Yaskawa INFORM job: DEMO_ROOF_UPPER_0625_3PAINT_42.JBI

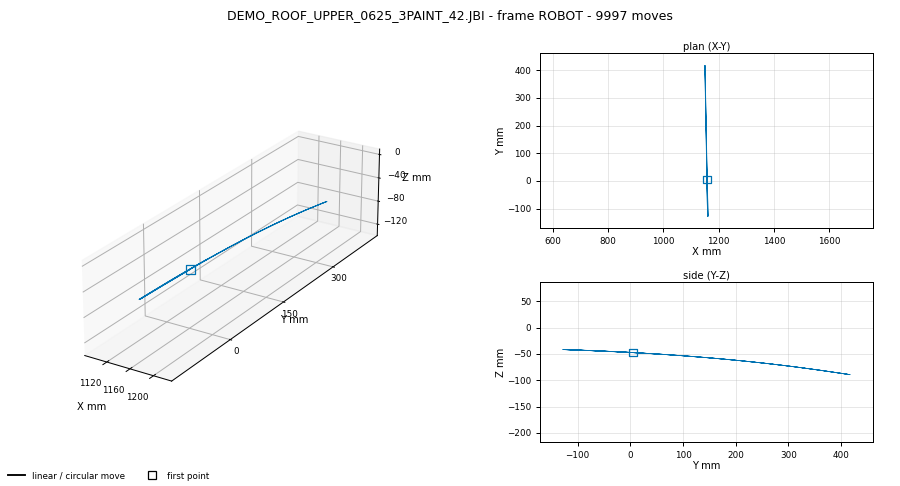
[picture p0: tool path of DEMO_ROOF_UPPER_0625_3PAINT_42.JBI in frame ROBOT, 9997 of 9997 moves have a stored position in this frame; points joined in program order, loops and branches not executed]
/JOB
//NAME DEMO_ROOF_UPPER_0625_3PAINT42
//POS
///NPOS 9997,0,0,0,0,0
///TOOL 0
///USER 0
///POSTYPE ROBOT
///RECTAN
///RCONF 1,0,0,0,0,0,0,0,0,0,0,0,0,0,0,0,0,0,0,0,0,0,0,0
C00000=1159.229,5.390,-47.328,179.872,6.067,149.128
C00001=1159.234,5.140,-47.313,179.870,6.066,149.128
C00002=1159.239,4.891,-47.300,179.867,6.066,149.129
C00003=1159.244,4.641,-47.286,179.865,6.065,149.129
C00004=1159.249,4.391,-47.273,179.863,6.064,149.130
C00005=1159.255,4.142,-47.259,179.860,6.063,149.131
C00006=1159.259,3.892,-47.246,179.858,6.063,149.131
C00007=1159.265,3.643,-47.232,179.855,6.061,149.132
C00008=1159.270,3.393,-47.218,179.852,6.061,149.132
C00009=1159.275,3.144,-47.205,179.850,6.060,149.133
C00010=1159.280,2.894,-47.192,179.848,6.060,149.134
C00011=1159.285,2.645,-47.178,179.845,6.059,149.134
C00012=1159.290,2.395,-47.165,179.843,6.058,149.135
C00013=1159.295,2.125,-47.150,179.840,6.058,149.135
C00014=1159.301,1.856,-47.135,179.837,6.057,149.136
C00015=1159.306,1.587,-47.121,179.835,6.056,149.137
C00016=1159.312,1.317,-47.106,179.832,6.055,149.137
C00017=1159.318,1.068,-47.093,179.829,6.055,149.138
C00018=1159.322,0.818,-47.080,179.827,6.054,149.138
C00019=1159.328,0.569,-47.066,179.824,6.053,149.139
C00020=1159.332,0.319,-47.053,179.822,6.052,149.140
C00021=1159.338,0.070,-47.039,179.819,6.052,149.140
C00022=1159.342,-0.180,-47.026,179.817,6.051,149.141
C00023=1159.348,-0.429,-47.013,179.814,6.050,149.141
C00024=1159.353,-0.680,-46.999,179.812,6.050,149.142
C00025=1159.358,-0.929,-46.986,179.809,6.049,149.143
C00026=1159.363,-1.179,-46.972,179.807,6.048,149.143
C00027=1159.368,-1.428,-46.960,179.805,6.048,149.144
C00028=1159.374,-1.678,-46.946,179.802,6.047,149.144
C00029=1159.379,-1.927,-46.933,179.799,6.046,149.145
C00030=1159.384,-2.177,-46.919,179.797,6.045,149.146
C00031=1159.389,-2.427,-46.906,179.794,6.044,149.146
C00032=1159.394,-2.676,-46.893,179.792,6.044,149.147
C00033=1159.399,-2.926,-46.880,179.790,6.043,149.147
C00034=1159.405,-3.175,-46.866,179.787,6.043,149.148
C00035=1159.410,-3.425,-46.854,179.785,6.042,149.148
C00036=1159.414,-3.674,-46.840,179.782,6.042,149.149
C00037=1159.420,-3.924,-46.827,179.780,6.041,149.150
C00038=1159.425,-4.174,-46.814,179.777,6.040,149.150
C00039=1159.430,-4.423,-46.801,179.775,6.039,149.151
C00040=1159.435,-4.673,-46.787,179.772,6.039,149.151
C00041=1159.441,-4.922,-46.774,179.770,6.039,149.152
C00042=1159.446,-5.172,-46.761,179.767,6.037,149.153
C00043=1159.450,-5.422,-46.748,179.764,6.036,149.153
C00044=1159.456,-5.671,-46.735,179.762,6.036,149.154
C00045=1159.460,-5.921,-46.721,179.759,6.035,149.154
C00046=1159.466,-6.170,-46.708,179.757,6.034,149.155
C00047=1159.471,-6.420,-46.696,179.755,6.034,149.156
C00048=1159.476,-6.670,-46.683,179.752,6.033,149.156
C00049=1159.482,-6.919,-46.669,179.750,6.033,149.157
C00050=1159.487,-7.169,-46.657,179.748,6.032,149.157
C00051=1159.492,-7.419,-46.643,179.745,6.031,149.158
C00052=1159.497,-7.668,-46.630,179.743,6.031,149.158
C00053=1159.502,-7.917,-46.617,179.740,6.030,149.159
C00054=1159.507,-8.167,-46.604,179.738,6.030,149.160
C00055=1159.512,-8.417,-46.591,179.735,6.029,149.160
C00056=1159.517,-8.667,-46.578,179.733,6.028,149.161
C00057=1159.523,-8.916,-46.565,179.731,6.028,149.161
C00058=1159.528,-9.166,-46.552,179.728,6.027,149.162
C00059=1159.532,-9.416,-46.540,179.726,6.026,149.162
C00060=1159.538,-9.665,-46.526,179.722,6.025,149.163
C00061=1159.543,-9.915,-46.514,179.720,6.024,149.164
C00062=1159.548,-10.165,-46.501,179.718,6.024,149.164
C00063=1159.554,-10.414,-46.488,179.715,6.023,149.165
C00064=1159.559,-10.664,-46.475,179.713,6.023,149.165
C00065=1159.564,-10.913,-46.462,179.711,6.022,149.166
C00066=1159.569,-11.163,-46.449,179.708,6.021,149.167
C00067=1159.574,-11.413,-46.436,179.705,6.021,149.167
C00068=1159.579,-11.662,-46.424,179.703,6.020,149.168
C00069=1159.584,-11.912,-46.411,179.700,6.020,149.168
C00070=1159.589,-12.161,-46.398,179.698,6.019,149.169
C00071=1159.595,-12.411,-46.385,179.696,6.018,149.170
C00072=1159.600,-12.661,-46.372,179.693,6.018,149.170
C00073=1159.605,-12.910,-46.359,179.691,6.017,149.171
C00074=1159.610,-13.159,-46.347,179.689,6.016,149.171
C00075=1159.616,-13.409,-46.333,179.686,6.016,149.172
C00076=1159.620,-13.659,-46.320,179.684,6.015,149.172
C00077=1159.625,-13.908,-46.308,179.681,6.015,149.173
C00078=1159.630,-14.158,-46.295,179.679,6.014,149.174
C00079=1159.636,-14.407,-46.283,179.676,6.013,149.174
C00080=1159.641,-14.657,-46.269,179.674,6.013,149.175
C00081=1159.646,-14.907,-46.257,179.671,6.012,149.175
C00082=1159.651,-15.157,-46.245,179.669,6.012,149.176
C00083=1159.656,-15.406,-46.232,179.667,6.011,149.177
C00084=1159.661,-15.656,-46.219,179.664,6.010,149.177
C00085=1159.667,-15.906,-46.206,179.662,6.010,149.178
C00086=1159.672,-16.155,-46.193,179.659,6.009,149.178
C00087=1159.677,-16.404,-46.181,179.657,6.008,149.179
C00088=1159.683,-16.654,-46.169,179.654,6.008,149.180
C00089=1159.687,-16.904,-46.156,179.652,6.007,149.180
C00090=1159.692,-17.154,-46.143,179.649,6.007,149.181
C00091=1159.697,-17.403,-46.131,179.647,6.006,149.181
C00092=1159.703,-17.652,-46.117,179.645,6.006,149.182
C00093=1159.708,-17.903,-46.105,179.642,6.005,149.183
C00094=1159.713,-18.152,-46.093,179.640,6.004,149.183
C00095=1159.718,-18.402,-46.080,179.637,6.004,149.184
C00096=1159.723,-18.651,-46.067,179.635,6.003,149.184
C00097=1159.728,-18.900,-46.055,179.632,6.003,149.185
C00098=1159.734,-19.150,-46.043,179.630,6.002,149.185
C00099=1159.738,-19.400,-46.030,179.627,6.001,149.186
C00100=1159.744,-19.650,-46.017,179.625,6.001,149.187
C00101=1159.750,-19.900,-46.005,179.623,6.000,149.187
C00102=1159.755,-20.149,-45.992,179.620,5.999,149.188
C00103=1159.760,-20.399,-45.980,179.618,5.999,149.188
C00104=1159.765,-20.648,-45.967,179.616,5.998,149.189
C00105=1159.770,-20.899,-45.955,179.613,5.998,149.190
C00106=1159.775,-21.148,-45.942,179.611,5.997,149.190
C00107=1159.780,-21.397,-45.930,179.608,5.996,149.191
C00108=1159.786,-21.647,-45.918,179.605,5.996,149.191
C00109=1159.791,-21.896,-45.905,179.603,5.995,149.192
C00110=1159.796,-22.146,-45.893,179.601,5.995,149.193
C00111=1159.801,-22.396,-45.881,179.598,5.994,149.193
C00112=1159.806,-22.645,-45.868,179.596,5.993,149.194
C00113=1159.811,-22.896,-45.856,179.594,5.993,149.194
C00114=1159.816,-23.145,-45.843,179.591,5.992,149.195
C00115=1159.821,-23.394,-45.831,179.589,5.991,149.195
C00116=1159.827,-23.644,-45.819,179.586,5.991,149.196
C00117=1159.832,-23.914,-45.805,179.583,5.991,149.197
C00118=1159.839,-24.184,-45.792,179.581,5.990,149.197
C00119=1159.844,-24.454,-45.778,179.578,5.989,149.198
C00120=1159.849,-24.723,-45.766,179.576,5.989,149.199
C00121=1159.854,-24.973,-45.753,179.574,5.988,149.199
C00122=1159.859,-25.223,-45.741,179.571,5.988,149.200
C00123=1159.865,-25.473,-45.728,179.569,5.987,149.200
C00124=1159.870,-25.722,-45.716,179.566,5.986,149.201
C00125=1159.875,-25.972,-45.704,179.564,5.986,149.202
C00126=1159.881,-26.222,-45.692,179.561,5.985,149.202
C00127=1159.886,-26.471,-45.679,179.559,5.985,149.203
C00128=1159.891,-26.721,-45.667,179.556,5.984,149.203
C00129=1159.896,-26.970,-45.655,179.554,5.984,149.204
C00130=1159.902,-27.220,-45.643,179.552,5.983,149.205
C00131=1159.906,-27.469,-45.631,179.549,5.982,149.205
C00132=1159.911,-27.719,-45.619,179.547,5.982,149.206
C00133=1159.917,-27.968,-45.606,179.545,5.982,149.206
C00134=1159.922,-28.218,-45.594,179.543,5.981,149.207
C00135=1159.927,-28.468,-45.582,179.540,5.981,149.208
C00136=1159.932,-28.718,-45.569,179.538,5.980,149.208
C00137=1159.937,-28.968,-45.558,179.535,5.979,149.209
C00138=1159.943,-29.218,-45.545,179.533,5.979,149.209
C00139=1159.948,-29.468,-45.533,179.530,5.978,149.210
C00140=1159.952,-29.717,-45.521,179.528,5.977,149.210
C00141=1159.958,-29.967,-45.509,179.525,5.977,149.211
C00142=1159.963,-30.216,-45.497,179.523,5.977,149.212
C00143=1159.968,-30.466,-45.485,179.520,5.976,149.212
C00144=1159.974,-30.716,-45.473,179.518,5.975,149.213
C00145=1159.979,-30.965,-45.460,179.516,5.974,149.213
C00146=1159.984,-31.215,-45.449,179.513,5.974,149.214
C00147=1159.989,-31.465,-45.437,179.511,5.974,149.215
C00148=1159.994,-31.714,-45.424,179.509,5.974,149.215
C00149=1160.000,-31.964,-45.413,179.507,5.973,149.216
C00150=1160.005,-32.214,-45.401,179.504,5.972,149.216
C00151=1160.009,-32.463,-45.389,179.502,5.972,149.217
C00152=1160.015,-32.713,-45.377,179.499,5.971,149.218
C00153=1160.020,-32.963,-45.365,179.497,5.970,149.218
C00154=1160.025,-33.212,-45.352,179.494,5.970,149.219
C00155=1160.031,-33.461,-45.341,179.492,5.969,149.219
C00156=1160.036,-33.711,-45.330,179.489,5.969,149.220
C00157=1160.041,-33.961,-45.318,179.487,5.968,149.220
C00158=1160.047,-34.210,-45.305,179.485,5.968,149.221
C00159=1160.052,-34.460,-45.293,179.483,5.967,149.222
C00160=1160.057,-34.710,-45.282,179.480,5.967,149.222
C00161=1160.062,-34.960,-45.270,179.478,5.967,149.223
C00162=1160.067,-35.209,-45.257,179.475,5.966,149.223
C00163=1160.073,-35.459,-45.246,179.473,5.965,149.224
C00164=1160.077,-35.708,-45.234,179.471,5.965,149.225
C00165=1160.083,-35.958,-45.222,179.468,5.964,149.225
C00166=1160.088,-36.208,-45.210,179.466,5.963,149.226
C00167=1160.093,-36.457,-45.198,179.463,5.963,149.227
C00168=1160.098,-36.707,-45.187,179.461,5.963,149.227
C00169=1160.104,-36.957,-45.175,179.459,5.963,149.228
C00170=1160.110,-37.206,-45.163,179.457,5.962,149.228
C00171=1160.114,-37.456,-45.152,179.454,5.961,149.229
C00172=1160.119,-37.705,-45.139,179.452,5.961,149.229
C00173=1160.125,-37.955,-45.127,179.449,5.960,149.230
C00174=1160.129,-38.205,-45.116,179.447,5.959,149.231
C00175=1160.135,-38.455,-45.104,179.444,5.959,149.231
C00176=1160.140,-38.705,-45.092,179.442,5.958,149.232
C00177=1160.145,-38.954,-45.081,179.440,5.958,149.232
C00178=1160.151,-39.204,-45.069,179.438,5.958,149.233
C00179=1160.156,-39.454,-45.058,179.435,5.957,149.234
C00180=1160.161,-39.703,-45.046,179.433,5.956,149.234
C00181=1160.166,-39.953,-45.034,179.430,5.956,149.235
C00182=1160.171,-40.202,-45.022,179.428,5.955,149.235
C00183=1160.176,-40.452,-45.011,179.425,5.955,149.236
C00184=1160.182,-40.702,-44.999,179.423,5.954,149.237
C00185=1160.187,-40.951,-44.988,179.421,5.954,149.237
C00186=1160.193,-41.201,-44.976,179.419,5.954,149.238
C00187=1160.198,-41.451,-44.964,179.416,5.953,149.238
C00188=1160.203,-41.700,-44.953,179.414,5.953,149.239
C00189=1160.208,-41.950,-44.941,179.412,5.952,149.239
C00190=1160.213,-42.200,-44.930,179.409,5.952,149.240
C00191=1160.218,-42.450,-44.918,179.407,5.951,149.241
C00192=1160.224,-42.699,-44.907,179.404,5.950,149.241
C00193=1160.229,-42.949,-44.895,179.402,5.950,149.242
C00194=1160.234,-43.199,-44.883,179.400,5.950,149.243
C00195=1160.239,-43.448,-44.872,179.398,5.949,149.243
C00196=1160.245,-43.698,-44.860,179.395,5.949,149.244
C00197=1160.250,-43.947,-44.849,179.393,5.948,149.244
C00198=1160.255,-44.197,-44.837,179.390,5.948,149.245
C00199=1160.260,-44.447,-44.826,179.388,5.947,149.245
C00200=1160.265,-44.697,-44.814,179.386,5.947,149.246
C00201=1160.270,-44.946,-44.802,179.384,5.946,149.247
C00202=1160.276,-45.196,-44.791,179.381,5.946,149.247
C00203=1160.281,-45.445,-44.780,179.379,5.945,149.248
C00204=1160.286,-45.695,-44.768,179.376,5.945,149.248
C00205=1160.291,-45.945,-44.757,179.374,5.944,149.249
C00206=1160.297,-46.195,-44.745,179.372,5.944,149.250
C00207=1160.302,-46.444,-44.734,179.370,5.943,149.250
C00208=1160.307,-46.694,-44.723,179.367,5.943,149.251
C00209=1160.312,-46.944,-44.711,179.365,5.942,149.251
C00210=1160.317,-47.194,-44.699,179.362,5.942,149.252
C00211=1160.323,-47.443,-44.688,179.360,5.941,149.252
C00212=1160.328,-47.693,-44.677,179.358,5.941,149.253
C00213=1160.333,-47.943,-44.666,179.356,5.941,149.254
C00214=1160.339,-48.193,-44.654,179.353,5.940,149.254
C00215=1160.344,-48.442,-44.643,179.351,5.939,149.255
C00216=1160.349,-48.691,-44.632,179.348,5.939,149.255
C00217=1160.354,-48.941,-44.620,179.346,5.938,149.256
C00218=1160.359,-49.190,-44.609,179.344,5.939,149.257
C00219=1160.365,-49.441,-44.598,179.342,5.938,149.257
C00220=1160.370,-49.690,-44.587,179.339,5.937,149.258
C00221=1160.375,-49.961,-44.574,179.336,5.937,149.259
C00222=1160.381,-50.231,-44.562,179.334,5.936,149.259
C00223=1160.387,-50.502,-44.549,179.332,5.936,149.260
C00224=1160.393,-50.772,-44.538,179.329,5.935,149.260
C00225=1160.398,-51.022,-44.526,179.327,5.935,149.261
C00226=1160.403,-51.272,-44.515,179.324,5.934,149.262
C00227=1160.408,-51.522,-44.504,179.322,5.934,149.262
C00228=1160.414,-51.771,-44.493,179.320,5.934,149.263
C00229=1160.419,-52.021,-44.481,179.318,5.933,149.263
C00230=1160.424,-52.271,-44.470,179.315,5.933,149.264
C00231=1160.429,-52.520,-44.460,179.313,5.932,149.264
C00232=1160.435,-52.770,-44.448,179.310,5.931,149.265
C00233=1160.439,-53.020,-44.436,179.308,5.931,149.266
C00234=1160.445,-53.269,-44.426,179.306,5.931,149.266
C00235=1160.450,-53.519,-44.414,179.304,5.930,149.267
C00236=1160.455,-53.769,-44.403,179.301,5.930,149.268
C00237=1160.461,-54.018,-44.393,179.299,5.929,149.268
C00238=1160.466,-54.268,-44.381,179.297,5.929,149.269
C00239=1160.471,-54.518,-44.370,179.294,5.929,149.269
C00240=1160.476,-54.767,-44.359,179.292,5.928,149.270
C00241=1160.481,-55.017,-44.348,179.290,5.927,149.270
C00242=1160.487,-55.268,-44.337,179.287,5.927,149.271
C00243=1160.492,-55.517,-44.326,179.285,5.927,149.272
C00244=1160.497,-55.766,-44.315,179.283,5.927,149.272
C00245=1160.503,-56.017,-44.304,179.281,5.926,149.273
C00246=1160.508,-56.266,-44.293,179.278,5.925,149.273
C00247=1160.513,-56.515,-44.281,179.276,5.925,149.274
C00248=1160.518,-56.765,-44.271,179.274,5.925,149.275
C00249=1160.524,-57.015,-44.259,179.271,5.924,149.275
C00250=1160.529,-57.265,-44.249,179.269,5.924,149.276
C00251=1160.534,-57.514,-44.238,179.267,5.923,149.276
C00252=1160.539,-57.764,-44.227,179.264,5.922,149.277
C00253=1160.544,-58.014,-44.215,179.262,5.923,149.277
C00254=1160.550,-58.264,-44.205,179.260,5.922,149.278
C00255=1160.555,-58.513,-44.194,179.257,5.921,149.279
C00256=1160.560,-58.763,-44.184,179.255,5.921,149.279
C00257=1160.565,-59.012,-44.172,179.253,5.921,149.280
C00258=1160.570,-59.262,-44.160,179.251,5.920,149.280
C00259=1160.576,-59.512,-44.150,179.248,5.920,149.281
C00260=1160.581,-59.762,-44.139,179.246,5.919,149.281
C00261=1160.586,-60.011,-44.129,179.243,5.919,149.282
C00262=1160.591,-60.261,-44.118,179.242,5.919,149.283
C00263=1160.597,-60.511,-44.107,179.239,5.918,149.283
C00264=1160.602,-60.761,-44.096,179.237,5.918,149.284
C00265=1160.607,-61.010,-44.085,179.234,5.917,149.285
C00266=1160.613,-61.260,-44.075,179.233,5.917,149.285
C00267=1160.617,-61.510,-44.063,179.230,5.917,149.286
C00268=1160.623,-61.759,-44.053,179.228,5.916,149.286
C00269=1160.628,-62.009,-44.041,179.225,5.916,149.287
C00270=1160.634,-62.259,-44.031,179.224,5.916,149.287
C00271=1160.639,-62.509,-44.020,179.221,5.915,149.288
C00272=1160.644,-62.758,-44.009,179.219,5.914,149.289
C00273=1160.649,-63.008,-43.999,179.216,5.914,149.289
C00274=1160.654,-63.257,-43.988,179.215,5.914,149.290
C00275=1160.659,-63.507,-43.977,179.212,5.913,149.290
C00276=1160.664,-63.758,-43.967,179.210,5.913,149.291
C00277=1160.670,-64.007,-43.955,179.207,5.912,149.291
C00278=1160.675,-64.257,-43.945,179.205,5.912,149.292
C00279=1160.681,-64.506,-43.934,179.203,5.912,149.293
C00280=1160.686,-64.756,-43.923,179.201,5.911,149.293
C00281=1160.691,-65.006,-43.913,179.198,5.910,149.294
C00282=1160.696,-65.255,-43.902,179.196,5.910,149.295
C00283=1160.702,-65.505,-43.891,179.194,5.910,149.295
C00284=1160.707,-65.755,-43.881,179.191,5.910,149.296
C00285=1160.712,-66.005,-43.871,179.189,5.909,149.296
C00286=1160.717,-66.254,-43.859,179.187,5.909,149.297
C00287=1160.722,-66.504,-43.849,179.185,5.908,149.297
C00288=1160.727,-66.754,-43.839,179.182,5.908,149.298
C00289=1160.734,-67.003,-43.827,179.180,5.907,149.299
C00290=1160.739,-67.253,-43.817,179.179,5.907,149.299
C00291=1160.744,-67.503,-43.806,179.176,5.907,149.300
C00292=1160.750,-67.753,-43.796,179.174,5.906,149.300
C00293=1160.754,-68.002,-43.785,179.171,5.906,149.301
C00294=1160.760,-68.252,-43.775,179.169,5.906,149.301
C00295=1160.765,-68.502,-43.764,179.167,5.905,149.302
C00296=1160.771,-68.752,-43.754,179.165,5.905,149.303
C00297=1160.775,-69.001,-43.743,179.162,5.904,149.303
C00298=1160.781,-69.251,-43.732,179.160,5.904,149.304
C00299=1160.786,-69.501,-43.722,179.158,5.904,149.304
C00300=1160.791,-69.751,-43.712,179.155,5.903,149.305
C00301=1160.797,-70.000,-43.701,179.153,5.903,149.306
C00302=1160.802,-70.250,-43.690,179.151,5.903,149.306
C00303=1160.807,-70.499,-43.680,179.149,5.902,149.307
C00304=1160.812,-70.750,-43.669,179.146,5.901,149.307
C00305=1160.818,-70.999,-43.659,179.145,5.901,149.308
C00306=1160.823,-71.249,-43.648,179.142,5.901,149.309
C00307=1160.828,-71.498,-43.638,179.140,5.900,149.309
C00308=1160.834,-71.748,-43.627,179.137,5.900,149.310
C00309=1160.839,-71.998,-43.617,179.136,5.900,149.310
C00310=1160.844,-72.248,-43.607,179.133,5.899,149.311
C00311=1160.849,-72.497,-43.597,179.131,5.899,149.311
C00312=1160.854,-72.747,-43.586,179.129,5.899,149.312
C00313=1160.860,-72.997,-43.576,179.126,5.898,149.313
C00314=1160.865,-73.247,-43.566,179.124,5.898,149.313
C00315=1160.871,-73.496,-43.555,179.122,5.897,149.314
C00316=1160.876,-73.745,-43.544,179.120,5.897,149.314
C00317=1160.881,-73.996,-43.534,179.117,5.897,149.315
C00318=1160.886,-74.245,-43.524,179.115,5.896,149.315
C00319=1160.891,-74.495,-43.513,179.113,5.896,149.316
C00320=1160.897,-74.745,-43.503,179.111,5.896,149.317
C00321=1160.903,-74.994,-43.493,179.109,5.895,149.317
C00322=1160.908,-75.245,-43.482,179.106,5.894,149.318
C00323=1160.912,-75.494,-43.473,179.104,5.894,149.318
C00324=1160.918,-75.743,-43.462,179.102,5.894,149.319
C00325=1160.924,-76.015,-43.451,179.100,5.893,149.319
C00326=1160.929,-76.286,-43.440,179.097,5.893,149.320
C00327=1160.936,-76.557,-43.429,179.095,5.893,149.321
C00328=1160.941,-76.829,-43.418,179.093,5.893,149.321
C00329=1160.946,-77.078,-43.407,179.090,5.892,149.322
C00330=1160.951,-77.328,-43.397,179.088,5.891,149.323
C00331=1160.957,-77.578,-43.387,179.086,5.892,149.323
C00332=1160.963,-77.827,-43.377,179.083,5.891,149.324
C00333=1160.968,-78.078,-43.366,179.081,5.890,149.324
C00334=1160.973,-78.327,-43.356,179.079,5.891,149.325
C00335=1160.978,-78.576,-43.346,179.077,5.890,149.325
C00336=1160.983,-78.827,-43.336,179.074,5.889,149.326
C00337=1160.989,-79.076,-43.325,179.072,5.889,149.327
C00338=1160.994,-79.326,-43.315,179.070,5.889,149.327
C00339=1161.000,-79.575,-43.305,179.068,5.888,149.328
C00340=1161.004,-79.825,-43.295,179.066,5.887,149.328
C00341=1161.010,-80.075,-43.285,179.064,5.888,149.329
C00342=1161.016,-80.325,-43.275,179.061,5.887,149.329
C00343=1161.021,-80.575,-43.265,179.059,5.887,149.330
C00344=1161.026,-80.824,-43.255,179.057,5.887,149.331
C00345=1161.031,-81.074,-43.245,179.054,5.886,149.331
C00346=1161.037,-81.323,-43.235,179.052,5.886,149.332
C00347=1161.042,-81.574,-43.224,179.051,5.886,149.332
C00348=1161.047,-81.823,-43.214,179.048,5.885,149.333
C00349=1161.052,-82.073,-43.205,179.046,5.884,149.334
C00350=1161.057,-82.323,-43.194,179.044,5.885,149.334
C00351=1161.063,-82.573,-43.184,179.042,5.884,149.335
C00352=1161.068,-82.822,-43.175,179.039,5.883,149.335
C00353=1161.074,-83.072,-43.164,179.037,5.884,149.336
C00354=1161.079,-83.322,-43.154,179.035,5.883,149.336
C00355=1161.084,-83.572,-43.144,179.032,5.883,149.337
C00356=1161.089,-83.821,-43.135,179.031,5.883,149.338
C00357=1161.095,-84.071,-43.124,179.028,5.882,149.338
C00358=1161.100,-84.321,-43.114,179.026,5.881,149.339
C00359=1161.105,-84.570,-43.104,179.024,5.881,149.339
C00360=1161.111,-84.821,-43.095,179.022,5.881,149.340
C00361=1161.116,-85.070,-43.085,179.020,5.880,149.340
C00362=1161.121,-85.320,-43.075,179.017,5.881,149.341
C00363=1161.126,-85.570,-43.064,179.015,5.880,149.342
C00364=1161.132,-85.819,-43.054,179.013,5.879,149.342
C00365=1161.137,-86.069,-43.045,179.011,5.880,149.343
C00366=1161.142,-86.318,-43.035,179.009,5.879,149.343
C00367=1161.147,-86.569,-43.024,179.006,5.878,149.344
C00368=1161.153,-86.819,-43.016,179.005,5.878,149.345
C00369=1161.158,-87.068,-43.005,179.002,5.878,149.345
C00370=1161.164,-87.318,-42.995,179.000,5.878,149.346
C00371=1161.169,-87.567,-42.986,178.998,5.877,149.346
C00372=1161.174,-87.818,-42.976,178.995,5.877,149.347
C00373=1161.179,-88.067,-42.966,178.994,5.877,149.347
C00374=1161.184,-88.317,-42.956,178.992,5.876,149.348
C00375=1161.190,-88.567,-42.946,178.989,5.876,149.349
C00376=1161.195,-88.816,-42.937,178.987,5.876,149.349
C00377=1161.200,-89.066,-42.926,178.985,5.875,149.350
C00378=1161.206,-89.316,-42.917,178.982,5.875,149.350
C00379=1161.211,-89.566,-42.907,178.981,5.875,149.351
C00380=1161.217,-89.815,-42.897,178.978,5.874,149.351
C00381=1161.222,-90.065,-42.888,178.976,5.873,149.352
C00382=1161.227,-90.314,-42.878,178.974,5.873,149.352
C00383=1161.232,-90.564,-42.868,178.972,5.873,149.353
C00384=1161.238,-90.815,-42.858,178.970,5.873,149.354
C00385=1161.243,-91.064,-42.848,178.967,5.873,149.354
C00386=1161.248,-91.314,-42.839,178.965,5.872,149.355
C00387=1161.254,-91.564,-42.829,178.964,5.872,149.355
C00388=1161.259,-91.813,-42.819,178.961,5.872,149.356
C00389=1161.265,-92.063,-42.810,178.959,5.871,149.357
C00390=1161.269,-92.313,-42.800,178.957,5.871,149.357
C00391=1161.275,-92.563,-42.790,178.955,5.870,149.358
C00392=1161.280,-92.812,-42.781,178.953,5.870,149.358
C00393=1161.286,-93.062,-42.771,178.950,5.870,149.359
C00394=1161.290,-93.312,-42.762,178.948,5.869,149.359
C00395=1161.296,-93.562,-42.752,178.946,5.869,149.360
C00396=1161.301,-93.811,-42.743,178.944,5.869,149.361
C00397=1161.307,-94.061,-42.732,178.942,5.868,149.361
C00398=1161.312,-94.310,-42.723,178.940,5.868,149.362
C00399=1161.317,-94.561,-42.713,178.937,5.868,149.362
C00400=1161.322,-94.811,-42.704,178.936,5.868,149.363
C00401=1161.328,-95.060,-42.694,178.933,5.868,149.363
C00402=1161.333,-95.310,-42.685,178.931,5.867,149.364
C00403=1161.339,-95.559,-42.675,178.929,5.867,149.364
C00404=1161.344,-95.809,-42.666,178.927,5.866,149.365
C00405=1161.349,-96.059,-42.656,178.924,5.866,149.366
C00406=1161.354,-96.309,-42.647,178.923,5.866,149.366
C00407=1161.360,-96.559,-42.637,178.920,5.865,149.367
C00408=1161.365,-96.808,-42.628,178.919,5.865,149.367
C00409=1161.371,-97.058,-42.618,178.916,5.865,149.368
C00410=1161.376,-97.308,-42.608,178.914,5.864,149.369
C00411=1161.382,-97.558,-42.599,178.912,5.864,149.369
C00412=1161.386,-97.808,-42.589,178.909,5.864,149.370
C00413=1161.392,-98.058,-42.579,178.908,5.864,149.370
C00414=1161.397,-98.308,-42.571,178.906,5.863,149.371
C00415=1161.402,-98.557,-42.561,178.903,5.863,149.371
C00416=1161.408,-98.807,-42.551,178.901,5.863,149.372
C00417=1161.413,-99.056,-42.542,178.899,5.862,149.372
C00418=1161.419,-99.306,-42.532,178.897,5.862,149.373
C00419=1161.424,-99.556,-42.523,178.895,5.862,149.374
C00420=1161.429,-99.805,-42.514,178.893,5.861,149.374
C00421=1161.435,-100.056,-42.504,178.891,5.861,149.375
C00422=1161.440,-100.305,-42.495,178.888,5.860,149.375
C00423=1161.445,-100.555,-42.485,178.887,5.860,149.376
C00424=1161.451,-100.805,-42.476,178.884,5.860,149.376
C00425=1161.455,-101.054,-42.467,178.882,5.859,149.377
C00426=1161.461,-101.304,-42.457,178.880,5.859,149.377
C00427=1161.467,-101.554,-42.448,178.878,5.859,149.378
C00428=1161.471,-101.803,-42.439,178.876,5.859,149.379
C00429=1161.478,-102.076,-42.429,178.873,5.859,149.379
C00430=1161.483,-102.348,-42.418,178.871,5.858,149.380
C00431=1161.490,-102.619,-42.409,178.869,5.858,149.380
C00432=1161.495,-102.891,-42.398,178.867,5.858,149.381
C00433=1161.500,-103.141,-42.389,178.864,5.857,149.382
C00434=1161.506,-103.391,-42.380,178.863,5.857,149.382
C00435=1161.511,-103.641,-42.370,178.860,5.856,149.383
C00436=1161.516,-103.890,-42.361,178.858,5.856,149.383
C00437=1161.522,-104.141,-42.352,178.856,5.856,149.384
C00438=1161.527,-104.390,-42.342,178.854,5.855,149.384
C00439=1161.532,-104.640,-42.333,178.852,5.856,149.385
C00440=1161.538,-104.890,-42.324,178.850,5.855,149.386
C00441=1161.543,-105.140,-42.315,178.848,5.855,149.386
C00442=1161.548,-105.390,-42.306,178.845,5.855,149.387
C00443=1161.553,-105.639,-42.297,178.843,5.854,149.387
C00444=1161.559,-105.889,-42.287,178.842,5.854,149.388
C00445=1161.564,-106.139,-42.278,178.839,5.853,149.388
C00446=1161.569,-106.389,-42.269,178.837,5.854,149.389
C00447=1161.575,-106.638,-42.259,178.835,5.853,149.389
C00448=1161.580,-106.888,-42.250,178.834,5.853,149.390
C00449=1161.585,-107.138,-42.241,178.831,5.852,149.391
C00450=1161.590,-107.388,-42.232,178.829,5.852,149.391
C00451=1161.596,-107.638,-42.223,178.827,5.852,149.392
C00452=1161.602,-107.887,-42.214,178.824,5.851,149.392
C00453=1161.607,-108.136,-42.205,178.823,5.851,149.393
C00454=1161.612,-108.386,-42.196,178.821,5.851,149.393
C00455=1161.617,-108.636,-42.187,178.819,5.851,149.394
C00456=1161.623,-108.886,-42.177,178.816,5.850,149.394
C00457=1161.628,-109.136,-42.169,178.815,5.850,149.395
C00458=1161.634,-109.386,-42.160,178.812,5.850,149.396
C00459=1161.639,-109.636,-42.151,178.810,5.849,149.396
C00460=1161.645,-109.886,-42.141,178.808,5.849,149.397
C00461=1161.649,-110.135,-42.132,178.806,5.848,149.397
C00462=1161.655,-110.385,-42.123,178.804,5.849,149.398
C00463=1161.660,-110.634,-42.114,178.802,5.848,149.398
C00464=1161.666,-110.884,-42.105,178.800,5.848,149.399
C00465=1161.671,-111.134,-42.096,178.798,5.848,149.400
C00466=1161.677,-111.384,-42.087,178.796,5.848,149.400
C00467=1161.682,-111.634,-42.078,178.794,5.847,149.400
C00468=1161.687,-111.884,-42.069,178.792,5.846,149.401
C00469=1161.692,-112.133,-42.060,178.790,5.847,149.402
C00470=1161.697,-112.383,-42.051,178.787,5.846,149.402
C00471=1161.704,-112.633,-42.042,178.786,5.846,149.403
C00472=1161.709,-112.883,-42.033,178.783,5.846,149.403
C00473=1161.714,-113.132,-42.024,178.781,5.846,149.404
C00474=1161.719,-113.382,-42.015,178.779,5.845,149.404
C00475=1161.725,-113.632,-42.007,178.777,5.845,149.405
C00476=1161.730,-113.882,-41.998,178.775,5.844,149.406
C00477=1161.735,-114.132,-41.989,178.773,5.845,149.406
C00478=1161.741,-114.381,-41.980,178.771,5.844,149.407
C00479=1161.747,-114.631,-41.971,178.769,5.843,149.407
C00480=1161.752,-114.881,-41.962,178.767,5.843,149.408
C00481=1161.757,-115.131,-41.953,178.765,5.843,149.408
C00482=1161.762,-115.381,-41.944,178.763,5.843,149.409
C00483=1161.767,-115.631,-41.935,178.760,5.842,149.409
C00484=1161.773,-115.880,-41.927,178.759,5.842,149.410
C00485=1161.778,-116.130,-41.918,178.757,5.842,149.410
C00486=1161.783,-116.379,-41.909,178.755,5.842,149.411
C00487=1161.788,-116.629,-41.900,178.752,5.841,149.412
C00488=1161.794,-116.879,-41.890,178.751,5.841,149.412
C00489=1161.800,-117.129,-41.882,178.749,5.841,149.413
C00490=1161.805,-117.378,-41.873,178.747,5.841,149.413
C00491=1161.810,-117.628,-41.864,178.744,5.840,149.414
C00492=1161.816,-117.878,-41.855,178.743,5.840,149.414
C00493=1161.821,-118.129,-41.847,178.741,5.839,149.415
C00494=1161.827,-118.378,-41.839,178.738,5.840,149.415
C00495=1161.832,-118.628,-41.830,178.736,5.839,149.416
C00496=1161.837,-118.878,-41.821,178.735,5.839,149.416
C00497=1161.842,-119.127,-41.812,178.732,5.838,149.417
C00498=1161.848,-119.377,-41.803,178.730,5.838,149.418
C00499=1161.853,-119.626,-41.794,178.728,5.838,149.418
C00500=1161.858,-119.876,-41.785,178.726,5.837,149.419
C00501=1161.864,-120.127,-41.777,178.724,5.837,149.419
C00502=1161.869,-120.377,-41.768,178.722,5.837,149.420
C00503=1161.875,-120.626,-41.760,178.720,5.837,149.420
C00504=1161.880,-120.876,-41.751,178.718,5.836,149.421
C00505=1161.885,-121.125,-41.742,178.716,5.836,149.421
C00506=1161.890,-121.375,-41.733,178.714,5.836,149.422
C00507=1161.896,-121.626,-41.725,178.712,5.836,149.422
C00508=1161.902,-121.875,-41.716,178.710,5.835,149.423
C00509=1161.907,-122.125,-41.708,178.708,5.835,149.423
C00510=1161.912,-122.375,-41.699,178.706,5.835,149.424
C00511=1161.918,-122.624,-41.690,178.704,5.835,149.425
C00512=1161.923,-122.874,-41.682,178.702,5.834,149.425
C00513=1161.928,-123.124,-41.673,178.700,5.834,149.426
C00514=1161.933,-123.374,-41.664,178.697,5.834,149.426
C00515=1161.939,-123.623,-41.656,178.696,5.834,149.427
C00516=1161.945,-123.874,-41.647,178.694,5.833,149.427
C00517=1161.950,-124.123,-41.639,178.692,5.833,149.428
C00518=1161.955,-124.373,-41.630,178.690,5.832,149.428
C00519=1161.961,-124.622,-41.621,178.688,5.833,149.429
C00520=1161.966,-124.873,-41.614,178.686,5.832,149.429
C00521=1161.971,-125.122,-41.605,178.684,5.832,149.430
C00522=1161.977,-125.372,-41.596,178.682,5.831,149.430
C00523=1161.982,-125.621,-41.587,178.680,5.832,149.431
C00524=1161.987,-125.872,-41.579,178.678,5.831,149.432
C00525=1161.992,-126.122,-41.570,178.676,5.831,149.432
C00526=1161.998,-126.371,-41.562,178.674,5.830,149.433
C00527=1162.004,-126.621,-41.553,178.672,5.830,149.433
C00528=1162.009,-126.871,-41.545,178.669,5.830,149.434
C00529=1162.014,-127.120,-41.536,178.668,5.830,149.434
C00530=1162.019,-127.370,-41.528,178.666,5.829,149.435
C00531=1162.024,-127.620,-41.519,178.664,5.829,149.435
C00532=1162.030,-127.869,-41.511,178.662,5.829,149.436
C00533=1161.610,-127.881,-41.553,178.659,5.833,149.438
C00534=1161.604,-127.632,-41.561,178.660,5.833,149.437
C00535=1161.598,-127.382,-41.570,178.662,5.833,149.437
C00536=1161.593,-127.132,-41.578,178.664,5.833,149.436
C00537=1161.587,-126.882,-41.586,178.666,5.834,149.436
C00538=1161.582,-126.632,-41.595,178.668,5.834,149.435
C00539=1161.577,-126.382,-41.604,178.670,5.834,149.434
C00540=1161.571,-126.132,-41.612,178.672,5.834,149.434
C00541=1161.566,-125.883,-41.620,178.674,5.835,149.433
C00542=1161.561,-125.633,-41.629,178.676,5.835,149.433
C00543=1161.556,-125.383,-41.637,178.679,5.835,149.432
C00544=1161.550,-125.134,-41.646,178.680,5.835,149.432
C00545=1161.545,-124.884,-41.655,178.682,5.836,149.431
C00546=1161.540,-124.634,-41.664,178.684,5.836,149.431
C00547=1161.534,-124.384,-41.671,178.687,5.836,149.430
C00548=1161.528,-124.134,-41.680,178.688,5.836,149.430
C00549=1161.523,-123.884,-41.689,178.690,5.837,149.429
C00550=1161.518,-123.634,-41.697,178.692,5.837,149.429
C00551=1161.512,-123.385,-41.706,178.695,5.837,149.428
C00552=1161.507,-123.135,-41.715,178.696,5.837,149.427
C00553=1161.502,-122.885,-41.724,178.698,5.838,149.427
C00554=1161.496,-122.635,-41.733,178.700,5.838,149.426
C00555=1161.490,-122.385,-41.740,178.702,5.839,149.426
C00556=1161.485,-122.136,-41.749,178.704,5.838,149.425
C00557=1161.480,-121.886,-41.758,178.707,5.839,149.425
C00558=1161.476,-121.636,-41.767,178.708,5.839,149.424
C00559=1161.470,-121.387,-41.775,178.710,5.840,149.424
C00560=1161.464,-121.137,-41.783,178.712,5.840,149.423
C00561=1161.459,-120.887,-41.792,178.715,5.840,149.423
C00562=1161.454,-120.637,-41.801,178.716,5.840,149.422
C00563=1161.448,-120.388,-41.810,178.718,5.841,149.422
C00564=1161.443,-120.138,-41.818,178.720,5.841,149.421
C00565=1161.438,-119.887,-41.827,178.723,5.841,149.420
C00566=1161.432,-119.638,-41.836,178.724,5.841,149.420
C00567=1161.427,-119.388,-41.844,178.726,5.842,149.419
C00568=1161.421,-119.138,-41.854,178.729,5.842,149.419
C00569=1161.416,-118.888,-41.862,178.731,5.842,149.418
C00570=1161.410,-118.639,-41.871,178.732,5.842,149.418
C00571=1161.405,-118.389,-41.880,178.735,5.843,149.417
C00572=1161.400,-118.140,-41.889,178.737,5.843,149.417
C00573=1161.394,-117.889,-41.897,178.739,5.843,149.416
C00574=1161.389,-117.639,-41.906,178.740,5.843,149.416
C00575=1161.384,-117.389,-41.915,178.743,5.844,149.415
C00576=1161.379,-117.140,-41.924,178.745,5.845,149.414
C00577=1161.373,-116.890,-41.932,178.747,5.845,149.414
C00578=1161.368,-116.641,-41.941,178.749,5.845,149.413
C00579=1161.362,-116.391,-41.950,178.751,5.845,149.413
C00580=1161.357,-116.141,-41.959,178.753,5.846,149.412
C00581=1161.352,-115.891,-41.968,178.755,5.846,149.412
C00582=1161.346,-115.642,-41.976,178.757,5.846,149.411
C00583=1161.341,-115.392,-41.985,178.759,5.846,149.411
C00584=1161.335,-115.142,-41.995,178.761,5.847,149.410
C00585=1161.330,-114.892,-42.004,178.763,5.847,149.410
C00586=1161.325,-114.642,-42.012,178.765,5.847,149.409
C00587=1161.320,-114.392,-42.021,178.767,5.847,149.408
C00588=1161.314,-114.143,-42.030,178.770,5.848,149.408
C00589=1161.309,-113.893,-42.039,178.771,5.848,149.407
C00590=1161.304,-113.643,-42.048,178.773,5.848,149.407
C00591=1161.299,-113.394,-42.057,178.776,5.849,149.406
C00592=1161.293,-113.143,-42.066,178.778,5.849,149.406
C00593=1161.287,-112.894,-42.075,178.780,5.850,149.405
C00594=1161.282,-112.644,-42.084,178.782,5.849,149.405
C00595=1161.277,-112.395,-42.092,178.784,5.850,149.404
C00596=1161.271,-112.145,-42.101,178.786,5.850,149.404
C00597=1161.266,-111.895,-42.110,178.788,5.851,149.403
C00598=1161.260,-111.645,-42.120,178.790,5.850,149.402
C00599=1161.255,-111.395,-42.129,178.792,5.851,149.402
C00600=1161.250,-111.145,-42.138,178.794,5.851,149.401
C00601=1161.245,-110.895,-42.146,178.796,5.851,149.401
C00602=1161.239,-110.646,-42.155,178.799,5.852,149.400
C00603=1161.234,-110.396,-42.164,178.800,5.852,149.400
C00604=1161.228,-110.146,-42.173,178.802,5.853,149.399
C00605=1161.223,-109.896,-42.182,178.804,5.852,149.398
C00606=1161.218,-109.647,-42.192,178.807,5.853,149.398
C00607=1161.213,-109.397,-42.201,178.808,5.853,149.398
C00608=1161.208,-109.147,-42.210,178.811,5.853,149.397
C00609=1161.202,-108.897,-42.219,178.813,5.853,149.396
C00610=1161.197,-108.647,-42.228,178.815,5.854,149.396
C00611=1161.191,-108.397,-42.237,178.817,5.855,149.395
C00612=1161.186,-108.147,-42.246,178.819,5.855,149.395
C00613=1161.180,-107.898,-42.255,178.821,5.855,149.394
C00614=1161.175,-107.649,-42.265,178.823,5.855,149.394
C00615=1161.170,-107.399,-42.273,178.825,5.856,149.393
C00616=1161.164,-107.149,-42.282,178.827,5.856,149.392
C00617=1161.159,-106.899,-42.292,178.829,5.856,149.392
C00618=1161.153,-106.649,-42.301,178.832,5.857,149.391
C00619=1161.148,-106.399,-42.310,178.834,5.857,149.391
C00620=1161.143,-106.150,-42.319,178.836,5.858,149.390
C00621=1161.137,-105.900,-42.329,178.838,5.857,149.390
C00622=1161.132,-105.650,-42.338,178.840,5.858,149.389
C00623=1161.127,-105.400,-42.347,178.842,5.858,149.389
C00624=1161.122,-105.151,-42.356,178.844,5.858,149.388
C00625=1161.116,-104.901,-42.366,178.846,5.859,149.387
C00626=1161.111,-104.651,-42.375,178.848,5.859,149.387
C00627=1161.106,-104.401,-42.383,178.850,5.860,149.386
C00628=1161.100,-104.151,-42.394,178.852,5.859,149.386
C00629=1161.095,-103.902,-42.403,178.855,5.860,149.385
C00630=1161.090,-103.652,-42.411,178.856,5.860,149.385
C00631=1161.085,-103.402,-42.420,178.859,5.860,149.384
C00632=1161.079,-103.152,-42.431,178.861,5.861,149.384
C00633=1161.074,-102.902,-42.439,178.863,5.861,149.383
C00634=1161.068,-102.631,-42.449,178.865,5.862,149.382
C00635=1161.062,-102.359,-42.459,178.868,5.862,149.382
C00636=1161.056,-102.086,-42.470,178.870,5.862,149.381
C00637=1161.051,-101.815,-42.480,178.872,5.862,149.380
C00638=1161.045,-101.565,-42.489,178.874,5.863,149.380
C00639=1161.040,-101.315,-42.499,178.876,5.863,149.379
C00640=1161.035,-101.065,-42.508,178.879,5.863,149.379
C00641=1161.029,-100.815,-42.517,178.880,5.863,149.378
C00642=1161.024,-100.566,-42.527,178.882,5.864,149.378
C00643=1161.019,-100.316,-42.536,178.885,5.864,149.377
C00644=1161.014,-100.067,-42.546,178.887,5.864,149.377
C00645=1161.008,-99.817,-42.555,178.889,5.865,149.376
C00646=1161.003,-99.567,-42.564,178.891,5.865,149.375
C00647=1160.997,-99.317,-42.574,178.893,5.866,149.375
C00648=1160.992,-99.067,-42.583,178.895,5.866,149.374
C00649=1160.987,-98.818,-42.592,178.897,5.866,149.374
C00650=1160.981,-98.568,-42.602,178.900,5.867,149.373
C00651=1160.976,-98.318,-42.611,178.901,5.867,149.373
C00652=1160.970,-98.069,-42.621,178.904,5.867,149.372
C00653=1160.965,-97.819,-42.630,178.906,5.868,149.372
C00654=1160.959,-97.569,-42.640,178.908,5.868,149.371
C00655=1160.955,-97.319,-42.649,178.910,5.868,149.370
C00656=1160.949,-97.070,-42.658,178.912,5.868,149.370
C00657=1160.944,-96.819,-42.669,178.914,5.869,149.369
C00658=1160.939,-96.569,-42.678,178.917,5.869,149.369
C00659=1160.934,-96.320,-42.688,178.918,5.869,149.368
C00660=1160.928,-96.070,-42.697,178.921,5.870,149.367
C00661=1160.923,-95.821,-42.707,178.923,5.870,149.367
C00662=1160.918,-95.571,-42.716,178.925,5.870,149.366
C00663=1160.912,-95.321,-42.726,178.928,5.871,149.366
C00664=1160.907,-95.071,-42.735,178.929,5.871,149.365
C00665=1160.901,-94.822,-42.745,178.931,5.871,149.365
C00666=1160.896,-94.572,-42.754,178.934,5.872,149.364
C00667=1160.891,-94.322,-42.764,178.936,5.872,149.364
C00668=1160.885,-94.072,-42.773,178.938,5.873,149.363
C00669=1160.880,-93.822,-42.784,178.940,5.872,149.362
C00670=1160.875,-93.572,-42.793,178.942,5.873,149.362
C00671=1160.870,-93.323,-42.803,178.945,5.873,149.361
C00672=1160.864,-93.073,-42.812,178.946,5.873,149.361
C00673=1160.859,-92.823,-42.822,178.949,5.874,149.360
C00674=1160.854,-92.574,-42.831,178.951,5.874,149.360
C00675=1160.848,-92.324,-42.841,178.953,5.874,149.359
C00676=1160.843,-92.074,-42.850,178.955,5.875,149.359
C00677=1160.838,-91.824,-42.861,178.957,5.875,149.358
C00678=1160.833,-91.575,-42.870,178.959,5.876,149.357
C00679=1160.827,-91.325,-42.880,178.962,5.876,149.357
C00680=1160.822,-91.075,-42.890,178.964,5.876,149.356
C00681=1160.816,-90.825,-42.899,178.966,5.877,149.356
C00682=1160.811,-90.576,-42.909,178.968,5.877,149.355
C00683=1160.806,-90.326,-42.919,178.970,5.877,149.355
C00684=1160.801,-90.076,-42.928,178.972,5.878,149.354
C00685=1160.796,-89.826,-42.938,178.974,5.877,149.353
C00686=1160.790,-89.576,-42.948,178.977,5.878,149.353
C00687=1160.784,-89.327,-42.958,178.979,5.879,149.352
C00688=1160.779,-89.077,-42.967,178.981,5.879,149.352
C00689=1160.774,-88.827,-42.977,178.983,5.879,149.351
C00690=1160.769,-88.577,-42.987,178.986,5.880,149.350
C00691=1160.764,-88.328,-42.997,178.987,5.880,149.350
C00692=1160.758,-88.078,-43.007,178.990,5.880,149.349
C00693=1160.753,-87.828,-43.016,178.992,5.881,149.349
C00694=1160.747,-87.579,-43.026,178.994,5.881,149.348
C00695=1160.742,-87.330,-43.036,178.996,5.881,149.348
C00696=1160.737,-87.079,-43.046,178.999,5.882,149.347
C00697=1160.732,-86.829,-43.056,179.000,5.882,149.347
C00698=1160.727,-86.580,-43.066,179.003,5.882,149.346
C00699=1160.721,-86.330,-43.075,179.005,5.883,149.345
C00700=1160.716,-86.080,-43.086,179.007,5.883,149.345
C00701=1160.711,-85.830,-43.095,179.009,5.884,149.344
C00702=1160.705,-85.581,-43.106,179.011,5.884,149.344
C00703=1160.699,-85.331,-43.115,179.014,5.884,149.343
C00704=1160.695,-85.081,-43.125,179.016,5.885,149.343
C00705=1160.690,-84.831,-43.135,179.018,5.884,149.342
C00706=1160.684,-84.582,-43.145,179.020,5.885,149.341
C00707=1160.679,-84.332,-43.155,179.022,5.886,149.341
C00708=1160.673,-84.082,-43.165,179.024,5.885,149.340
C00709=1160.668,-83.832,-43.175,179.026,5.886,149.340
C00710=1160.663,-83.583,-43.185,179.029,5.887,149.339
C00711=1160.658,-83.333,-43.195,179.031,5.887,149.338
C00712=1160.652,-83.084,-43.205,179.033,5.887,149.338
C00713=1160.647,-82.833,-43.215,179.036,5.888,149.337
C00714=1160.642,-82.583,-43.225,179.037,5.888,149.337
C00715=1160.636,-82.334,-43.235,179.040,5.888,149.336
C00716=1160.631,-82.084,-43.245,179.042,5.889,149.336
C00717=1160.626,-81.834,-43.256,179.044,5.888,149.335
C00718=1160.621,-81.585,-43.265,179.046,5.889,149.334
C00719=1160.615,-81.335,-43.275,179.049,5.890,149.334
C00720=1160.609,-81.085,-43.285,179.051,5.890,149.333
C00721=1160.604,-80.835,-43.295,179.053,5.890,149.333
C00722=1160.600,-80.586,-43.305,179.055,5.891,149.332
C00723=1160.594,-80.336,-43.315,179.058,5.892,149.332
C00724=1160.589,-80.086,-43.326,179.059,5.891,149.331
C00725=1160.583,-79.836,-43.336,179.062,5.892,149.330
C00726=1160.579,-79.587,-43.346,179.064,5.893,149.330
C00727=1160.573,-79.338,-43.356,179.066,5.892,149.329
C00728=1160.568,-79.087,-43.366,179.068,5.893,149.329
C00729=1160.562,-78.837,-43.376,179.071,5.893,149.328
C00730=1160.556,-78.588,-43.386,179.073,5.893,149.328
C00731=1160.552,-78.338,-43.396,179.075,5.894,149.327
C00732=1160.547,-78.088,-43.406,179.078,5.895,149.326
C00733=1160.541,-77.839,-43.417,179.079,5.895,149.326
C00734=1160.536,-77.588,-43.427,179.082,5.895,149.325
C00735=1160.530,-77.339,-43.437,179.084,5.896,149.325
C00736=1160.525,-77.089,-43.448,179.086,5.895,149.324
C00737=1160.520,-76.839,-43.458,179.088,5.896,149.323
C00738=1160.514,-76.569,-43.469,179.091,5.896,149.323
C00739=1160.508,-76.297,-43.480,179.093,5.897,149.322
C00740=1160.503,-76.026,-43.491,179.096,5.898,149.322
C00741=1160.496,-75.755,-43.502,179.098,5.898,149.321
C00742=1160.492,-75.505,-43.512,179.100,5.898,149.320
C00743=1160.486,-75.255,-43.523,179.102,5.899,149.320
C00744=1160.481,-75.006,-43.533,179.105,5.899,149.319
C00745=1160.476,-74.755,-43.543,179.107,5.899,149.319
C00746=1160.470,-74.506,-43.554,179.109,5.900,149.318
C00747=1160.465,-74.256,-43.564,179.111,5.900,149.317
C00748=1160.460,-74.007,-43.575,179.113,5.900,149.317
C00749=1160.454,-73.757,-43.585,179.116,5.901,149.316
C00750=1160.449,-73.507,-43.596,179.118,5.902,149.316
C00751=1160.444,-73.257,-43.606,179.121,5.902,149.315
C00752=1160.438,-73.008,-43.616,179.122,5.902,149.315
C00753=1160.434,-72.758,-43.626,179.125,5.902,149.314
C00754=1160.428,-72.508,-43.636,179.127,5.903,149.313
C00755=1160.423,-72.259,-43.647,179.129,5.903,149.313
C00756=1160.418,-72.009,-43.657,179.131,5.903,149.312
C00757=1160.412,-71.759,-43.667,179.134,5.904,149.312
C00758=1160.407,-71.509,-43.679,179.136,5.905,149.311
C00759=1160.402,-71.260,-43.689,179.138,5.905,149.311
C00760=1160.396,-71.010,-43.699,179.140,5.905,149.310
C00761=1160.391,-70.760,-43.710,179.143,5.906,149.309
C00762=1160.386,-70.511,-43.720,179.145,5.906,149.309
C00763=1160.381,-70.260,-43.730,179.147,5.906,149.308
C00764=1160.375,-70.011,-43.741,179.149,5.907,149.307
C00765=1160.370,-69.761,-43.752,179.152,5.907,149.307
C00766=1160.365,-69.512,-43.762,179.154,5.907,149.306
C00767=1160.359,-69.262,-43.772,179.156,5.908,149.306
C00768=1160.354,-69.012,-43.783,179.158,5.909,149.305
C00769=1160.349,-68.763,-43.794,179.161,5.909,149.305
C00770=1160.344,-68.513,-43.804,179.162,5.909,149.304
C00771=1160.338,-68.263,-43.815,179.165,5.909,149.303
C00772=1160.333,-68.013,-43.825,179.167,5.910,149.303
C00773=1160.328,-67.764,-43.836,179.170,5.910,149.302
C00774=1160.323,-67.514,-43.847,179.171,5.910,149.302
C00775=1160.317,-67.264,-43.857,179.174,5.911,149.301
C00776=1160.312,-67.014,-43.868,179.176,5.912,149.301
C00777=1160.307,-66.765,-43.878,179.179,5.912,149.300
C00778=1160.302,-66.515,-43.889,179.181,5.912,149.299
C00779=1160.297,-66.265,-43.899,179.183,5.913,149.299
C00780=1160.291,-66.016,-43.910,179.185,5.913,149.298
C00781=1160.285,-65.766,-43.921,179.188,5.914,149.298
C00782=1160.280,-65.516,-43.932,179.190,5.914,149.297
C00783=1160.275,-65.266,-43.942,179.192,5.914,149.297
C00784=1160.270,-65.017,-43.953,179.195,5.915,149.296
C00785=1160.265,-64.767,-43.964,179.197,5.916,149.295
C00786=1160.259,-64.517,-43.974,179.199,5.915,149.295
C00787=1160.254,-64.268,-43.985,179.201,5.916,149.294
C00788=1160.249,-64.018,-43.995,179.204,5.916,149.293
C00789=1160.244,-63.768,-44.007,179.206,5.917,149.293
C00790=1160.238,-63.519,-44.017,179.208,5.917,149.292
C00791=1160.233,-63.268,-44.028,179.210,5.918,149.292
C00792=1160.228,-63.019,-44.039,179.213,5.918,149.291
C00793=1160.222,-62.769,-44.049,179.215,5.919,149.291
C00794=1160.217,-62.519,-44.060,179.217,5.919,149.290
C00795=1160.212,-62.270,-44.071,179.219,5.919,149.289
C00796=1160.207,-62.020,-44.082,179.221,5.920,149.289
C00797=1160.202,-61.771,-44.092,179.224,5.920,149.288
C00798=1160.197,-61.521,-44.103,179.226,5.920,149.288
C00799=1160.191,-61.271,-44.115,179.228,5.921,149.287
C00800=1160.186,-61.021,-44.125,179.231,5.921,149.287
C00801=1160.180,-60.772,-44.135,179.233,5.922,149.286
C00802=1160.176,-60.522,-44.147,179.235,5.922,149.285
C00803=1160.171,-60.272,-44.157,179.238,5.922,149.285
C00804=1160.164,-60.022,-44.169,179.240,5.923,149.284
C00805=1160.159,-59.772,-44.179,179.242,5.923,149.284
C00806=1160.154,-59.523,-44.190,179.245,5.924,149.283
C00807=1160.149,-59.273,-44.201,179.247,5.924,149.282
C00808=1160.144,-59.024,-44.212,179.249,5.925,149.282
C00809=1160.139,-58.774,-44.222,179.251,5.925,149.281
C00810=1160.133,-58.524,-44.234,179.254,5.926,149.281
C00811=1160.128,-58.274,-44.244,179.256,5.925,149.280
C00812=1160.123,-58.025,-44.256,179.258,5.926,149.280
C00813=1160.118,-57.775,-44.266,179.260,5.927,149.279
C00814=1160.112,-57.525,-44.278,179.263,5.927,149.278
C00815=1160.107,-57.276,-44.289,179.265,5.928,149.278
C00816=1160.102,-57.026,-44.299,179.267,5.928,149.277
C00817=1160.097,-56.776,-44.311,179.269,5.929,149.277
C00818=1160.091,-56.526,-44.322,179.272,5.929,149.276
C00819=1160.086,-56.277,-44.333,179.274,5.930,149.275
C00820=1160.081,-56.027,-44.343,179.277,5.930,149.275
C00821=1160.076,-55.778,-44.354,179.278,5.930,149.274
C00822=1160.070,-55.528,-44.366,179.281,5.931,149.274
C00823=1160.065,-55.278,-44.377,179.283,5.931,149.273
C00824=1160.060,-55.029,-44.388,179.286,5.932,149.272
C00825=1160.055,-54.779,-44.399,179.288,5.933,149.272
C00826=1160.050,-54.529,-44.410,179.290,5.932,149.271
C00827=1160.044,-54.280,-44.421,179.292,5.933,149.271
C00828=1160.040,-54.030,-44.432,179.295,5.933,149.270
C00829=1160.034,-53.779,-44.443,179.297,5.934,149.270
C00830=1160.029,-53.530,-44.454,179.300,5.935,149.269
C00831=1160.024,-53.281,-44.466,179.301,5.935,149.268
C00832=1160.018,-53.030,-44.477,179.304,5.935,149.268
C00833=1160.013,-52.781,-44.488,179.306,5.936,149.267
C00834=1160.008,-52.532,-44.499,179.309,5.936,149.267
C00835=1160.003,-52.281,-44.510,179.311,5.937,149.266
C00836=1159.997,-52.032,-44.521,179.313,5.937,149.265
C00837=1159.993,-51.783,-44.532,179.315,5.937,149.265
C00838=1159.987,-51.532,-44.544,179.318,5.938,149.264
C00839=1159.982,-51.282,-44.555,179.320,5.939,149.264
C00840=1159.976,-51.033,-44.566,179.323,5.939,149.263
C00841=1159.971,-50.784,-44.578,179.325,5.940,149.262
C00842=1159.966,-50.513,-44.590,179.328,5.940,149.262
C00843=1159.960,-50.242,-44.602,179.330,5.941,149.261
C00844=1159.954,-49.971,-44.614,179.332,5.941,149.261
C00845=1159.949,-49.702,-44.626,179.335,5.941,149.260
C00846=1159.943,-49.451,-44.637,179.337,5.942,149.259
C00847=1159.938,-49.202,-44.649,179.340,5.942,149.259
C00848=1159.933,-48.952,-44.660,179.342,5.943,149.258
C00849=1159.928,-48.703,-44.671,179.344,5.943,149.258
C00850=1159.922,-48.453,-44.683,179.347,5.944,149.257
C00851=1159.917,-48.203,-44.694,179.349,5.944,149.256
C00852=1159.913,-47.953,-44.705,179.351,5.945,149.256
C00853=1159.906,-47.704,-44.717,179.354,5.945,149.255
C00854=1159.902,-47.454,-44.728,179.356,5.946,149.255
C00855=1159.896,-47.204,-44.740,179.358,5.946,149.254
C00856=1159.892,-46.955,-44.751,179.361,5.947,149.253
C00857=1159.885,-46.705,-44.762,179.363,5.947,149.253
C00858=1159.881,-46.455,-44.773,179.365,5.947,149.252
C00859=1159.875,-46.205,-44.785,179.367,5.948,149.252
C00860=1159.871,-45.956,-44.796,179.370,5.948,149.251
C00861=1159.865,-45.706,-44.808,179.372,5.949,149.250
C00862=1159.860,-45.457,-44.819,179.375,5.949,149.250
C00863=1159.854,-45.207,-44.831,179.377,5.950,149.249
C00864=1159.850,-44.957,-44.842,179.379,5.950,149.249
C00865=1159.844,-44.708,-44.854,179.381,5.951,149.248
C00866=1159.839,-44.458,-44.865,179.384,5.951,149.247
C00867=1159.834,-44.209,-44.877,179.386,5.952,149.247
C00868=1159.829,-43.959,-44.888,179.389,5.952,149.246
C00869=1159.823,-43.708,-44.899,179.391,5.953,149.246
C00870=1159.818,-43.459,-44.910,179.394,5.953,149.245
C00871=1159.812,-43.209,-44.922,179.395,5.953,149.245
C00872=1159.807,-42.960,-44.934,179.398,5.954,149.244
C00873=1159.802,-42.710,-44.945,179.400,5.955,149.243
C00874=1159.797,-42.460,-44.957,179.403,5.955,149.243
C00875=1159.792,-42.210,-44.969,179.405,5.956,149.242
C00876=1159.786,-41.961,-44.980,179.408,5.956,149.242
C00877=1159.781,-41.711,-44.991,179.410,5.957,149.241
C00878=1159.776,-41.462,-45.003,179.412,5.957,149.240
C00879=1159.771,-41.212,-45.016,179.414,5.958,149.240
C00880=1159.766,-40.963,-45.027,179.417,5.958,149.239
C00881=1159.761,-40.713,-45.039,179.419,5.959,149.239
C00882=1159.755,-40.464,-45.050,179.422,5.959,149.238
C00883=1159.750,-40.214,-45.062,179.424,5.960,149.238
C00884=1159.745,-39.964,-45.074,179.427,5.960,149.237
C00885=1159.740,-39.714,-45.085,179.429,5.961,149.236
C00886=1159.734,-39.464,-45.097,179.431,5.961,149.236
C00887=1159.729,-39.214,-45.109,179.433,5.962,149.235
C00888=1159.724,-38.965,-45.120,179.436,5.962,149.234
C00889=1159.718,-38.715,-45.132,179.438,5.963,149.234
C00890=1159.713,-38.466,-45.144,179.441,5.963,149.233
C00891=1159.709,-38.217,-45.156,179.443,5.964,149.233
C00892=1159.703,-37.967,-45.167,179.445,5.964,149.232
C00893=1159.698,-37.717,-45.179,179.448,5.965,149.232
C00894=1159.693,-37.467,-45.191,179.450,5.966,149.231
C00895=1159.688,-37.217,-45.202,179.452,5.966,149.230
C00896=1159.682,-36.967,-45.214,179.454,5.966,149.230
C00897=1159.677,-36.718,-45.226,179.457,5.967,149.229
C00898=1159.672,-36.468,-45.238,179.459,5.967,149.229
C00899=1159.666,-36.219,-45.250,179.462,5.968,149.228
C00900=1159.662,-35.969,-45.261,179.464,5.969,149.227
C00901=1159.656,-35.719,-45.273,179.467,5.969,149.227
C00902=1159.651,-35.470,-45.285,179.469,5.970,149.226
C00903=1159.646,-35.220,-45.297,179.472,5.970,149.226
C00904=1159.641,-34.971,-45.309,179.474,5.971,149.225
C00905=1159.635,-34.721,-45.321,179.476,5.971,149.224
C00906=1159.630,-34.471,-45.333,179.478,5.971,149.224
C00907=1159.625,-34.221,-45.345,179.481,5.972,149.223
C00908=1159.620,-33.972,-45.356,179.483,5.973,149.223
C00909=1159.615,-33.722,-45.368,179.486,5.973,149.222
C00910=1159.609,-33.472,-45.380,179.488,5.974,149.222
C00911=1159.604,-33.223,-45.393,179.490,5.974,149.221
C00912=1159.600,-32.973,-45.404,179.493,5.975,149.220
C00913=1159.594,-32.723,-45.416,179.495,5.975,149.220
C00914=1159.589,-32.474,-45.429,179.497,5.976,149.219
C00915=1159.584,-32.224,-45.440,179.500,5.977,149.219
C00916=1159.578,-31.974,-45.452,179.502,5.977,149.218
C00917=1159.574,-31.725,-45.464,179.504,5.977,149.217
C00918=1159.568,-31.476,-45.476,179.507,5.978,149.217
C00919=1159.562,-31.226,-45.488,179.509,5.978,149.216
C00920=1159.557,-30.976,-45.500,179.511,5.979,149.216
C00921=1159.552,-30.726,-45.512,179.514,5.980,149.215
C00922=1159.547,-30.477,-45.524,179.517,5.980,149.214
C00923=1159.542,-30.227,-45.536,179.519,5.981,149.214
C00924=1159.536,-29.977,-45.548,179.522,5.981,149.213
C00925=1159.532,-29.727,-45.561,179.524,5.982,149.213
C00926=1159.527,-29.478,-45.573,179.526,5.982,149.212
C00927=1159.521,-29.228,-45.585,179.529,5.983,149.212
C00928=1159.516,-28.978,-45.597,179.531,5.984,149.211
C00929=1159.511,-28.729,-45.609,179.533,5.985,149.210
C00930=1159.506,-28.479,-45.621,179.536,5.984,149.210
C00931=1159.501,-28.229,-45.633,179.538,5.985,149.209
C00932=1159.496,-27.980,-45.646,179.540,5.985,149.208
C00933=1159.490,-27.730,-45.658,179.543,5.986,149.208
C00934=1159.485,-27.480,-45.669,179.545,5.987,149.207
C00935=1159.480,-27.231,-45.682,179.547,5.987,149.207
C00936=1159.474,-26.981,-45.694,179.550,5.988,149.206
C00937=1159.469,-26.732,-45.707,179.552,5.989,149.206
C00938=1159.464,-26.482,-45.718,179.555,5.989,149.205
C00939=1159.459,-26.233,-45.730,179.557,5.990,149.204
C00940=1159.454,-25.983,-45.742,179.560,5.990,149.204
C00941=1159.449,-25.733,-45.755,179.562,5.991,149.203
C00942=1159.443,-25.484,-45.767,179.565,5.992,149.203
C00943=1159.438,-25.234,-45.779,179.567,5.992,149.202
C00944=1159.434,-24.984,-45.792,179.569,5.993,149.201
C00945=1159.428,-24.734,-45.804,179.572,5.993,149.201
C00946=1159.423,-24.465,-45.818,179.574,5.994,149.200
C00947=1159.417,-24.195,-45.831,179.577,5.994,149.200
C00948=1159.411,-23.924,-45.844,179.580,5.995,149.199
C00949=1159.406,-23.655,-45.857,179.582,5.995,149.198
C00950=1159.400,-23.405,-45.869,179.584,5.996,149.198
C00951=1159.395,-23.156,-45.882,179.587,5.997,149.197
C00952=1159.391,-22.906,-45.895,179.589,5.997,149.197
C00953=1159.385,-22.656,-45.907,179.592,5.998,149.196
C00954=1159.380,-22.407,-45.919,179.594,5.999,149.195
C00955=1159.375,-22.157,-45.932,179.597,5.999,149.195
C00956=1159.369,-21.907,-45.944,179.599,6.000,149.194
C00957=1159.364,-21.658,-45.956,179.602,6.000,149.194
C00958=1159.359,-21.409,-45.969,179.604,6.001,149.193
C00959=1159.354,-21.159,-45.981,179.606,6.001,149.192
C00960=1159.349,-20.909,-45.994,179.609,6.002,149.192
C00961=1159.344,-20.659,-46.007,179.611,6.003,149.191
C00962=1159.338,-20.409,-46.019,179.614,6.003,149.191
C00963=1159.333,-20.160,-46.032,179.616,6.004,149.190
C00964=1159.328,-19.911,-46.044,179.619,6.004,149.189
C00965=1159.322,-19.661,-46.056,179.621,6.005,149.189
C00966=1159.317,-19.411,-46.069,179.624,6.006,149.188
C00967=1159.313,-19.161,-46.082,179.626,6.006,149.188
C00968=1159.308,-18.912,-46.094,179.628,6.007,149.187
C00969=1159.302,-18.662,-46.106,179.631,6.008,149.187
C00970=1159.297,-18.413,-46.119,179.633,6.008,149.186
C00971=1159.292,-18.163,-46.131,179.635,6.009,149.185
C00972=1159.287,-17.913,-46.144,179.638,6.009,149.185
C00973=1159.281,-17.663,-46.157,179.640,6.010,149.184
C00974=1159.276,-17.414,-46.169,179.643,6.011,149.184
C00975=1159.271,-17.165,-46.182,179.645,6.011,149.183
C00976=1159.266,-16.915,-46.195,179.648,6.012,149.182
C00977=1159.261,-16.665,-46.208,179.650,6.012,149.182
C00978=1159.256,-16.415,-46.219,179.653,6.013,149.181
C00979=1159.251,-16.166,-46.232,179.655,6.014,149.181
C00980=1159.245,-15.916,-46.245,179.658,6.014,149.180
C00981=1159.240,-15.667,-46.258,179.660,6.015,149.179
C00982=1159.235,-15.417,-46.271,179.662,6.016,149.179
C00983=1159.230,-15.168,-46.283,179.665,6.016,149.178
C00984=1159.225,-14.918,-46.295,179.667,6.017,149.178
C00985=1159.219,-14.668,-46.308,179.670,6.017,149.177
C00986=1159.214,-14.418,-46.321,179.672,6.018,149.177
C00987=1159.209,-14.169,-46.334,179.675,6.019,149.176
C00988=1159.204,-13.919,-46.347,179.677,6.019,149.175
C00989=1159.199,-13.670,-46.359,179.680,6.020,149.175
C00990=1159.194,-13.420,-46.373,179.682,6.020,149.174
C00991=1159.188,-13.170,-46.385,179.684,6.021,149.174
C00992=1159.183,-12.921,-46.398,179.687,6.021,149.173
C00993=1159.178,-12.672,-46.411,179.689,6.022,149.172
C00994=1159.174,-12.422,-46.424,179.692,6.023,149.172
C00995=1159.168,-12.172,-46.437,179.694,6.024,149.171
C00996=1159.163,-11.923,-46.449,179.697,6.024,149.171
C00997=1159.158,-11.673,-46.462,179.699,6.025,149.170
C00998=1159.152,-11.423,-46.476,179.702,6.025,149.169
C00999=1159.147,-11.174,-46.488,179.704,6.026,149.169
C01000=1159.143,-10.924,-46.501,179.706,6.026,149.168
C01001=1159.138,-10.675,-46.514,179.709,6.027,149.168
C01002=1159.132,-10.425,-46.527,179.711,6.028,149.167
C01003=1159.127,-10.176,-46.539,179.713,6.029,149.167
C01004=1159.122,-9.926,-46.552,179.716,6.029,149.166
C01005=1159.117,-9.676,-46.565,179.719,6.029,149.165
C01006=1159.111,-9.427,-46.578,179.721,6.030,149.165
C01007=1159.107,-9.177,-46.591,179.723,6.031,149.164
C01008=1159.101,-8.927,-46.604,179.726,6.032,149.164
C01009=1159.096,-8.678,-46.617,179.729,6.033,149.163
C01010=1159.091,-8.428,-46.630,179.731,6.034,149.162
C01011=1159.086,-8.178,-46.643,179.734,6.034,149.162
C01012=1159.081,-7.928,-46.656,179.736,6.035,149.161
C01013=1159.076,-7.679,-46.669,179.739,6.035,149.161
C01014=1159.070,-7.429,-46.681,179.741,6.036,149.160
C01015=1159.065,-7.180,-46.696,179.743,6.037,149.159
C01016=1159.060,-6.930,-46.708,179.746,6.037,149.159
C01017=1159.054,-6.681,-46.721,179.748,6.038,149.158
C01018=1159.050,-6.431,-46.734,179.751,6.038,149.158
C01019=1159.045,-6.181,-46.747,179.753,6.039,149.157
C01020=1159.039,-5.932,-46.760,179.756,6.039,149.156
C01021=1159.034,-5.682,-46.773,179.758,6.040,149.156
C01022=1159.029,-5.433,-46.787,179.761,6.041,149.155
C01023=1159.024,-5.183,-46.800,179.763,6.042,149.155
C01024=1159.019,-4.933,-46.813,179.765,6.042,149.154
C01025=1159.013,-4.684,-46.826,179.768,6.044,149.154
C01026=1159.009,-4.434,-46.839,179.771,6.044,149.153
C01027=1159.003,-4.185,-46.853,179.773,6.045,149.152
C01028=1158.999,-3.935,-46.866,179.776,6.045,149.152
C01029=1158.993,-3.685,-46.879,179.778,6.046,149.151
C01030=1158.988,-3.436,-46.891,179.780,6.047,149.151
C01031=1158.984,-3.186,-46.905,179.783,6.047,149.150
C01032=1158.978,-2.937,-46.918,179.785,6.048,149.149
C01033=1158.973,-2.687,-46.931,179.788,6.048,149.149
C01034=1158.967,-2.437,-46.945,179.790,6.049,149.148
C01035=1158.963,-2.188,-46.958,179.793,6.050,149.148
C01036=1158.957,-1.938,-46.971,179.795,6.050,149.147
C01037=1158.952,-1.689,-46.984,179.798,6.052,149.146
C01038=1158.947,-1.439,-46.998,179.800,6.052,149.146
C01039=1158.942,-1.190,-47.011,179.803,6.053,149.145
C01040=1158.937,-0.939,-47.024,179.805,6.054,149.145
C01041=1158.932,-0.691,-47.038,179.808,6.054,149.144
C01042=1158.927,-0.440,-47.051,179.810,6.055,149.144
C01043=1158.921,-0.191,-47.065,179.813,6.055,149.143
C01044=1158.917,0.059,-47.078,179.815,6.056,149.143
C01045=1158.911,0.308,-47.091,179.818,6.057,149.142
C01046=1158.907,0.558,-47.105,179.820,6.058,149.141
C01047=1158.901,0.807,-47.118,179.823,6.059,149.141
C01048=1158.896,1.057,-47.131,179.826,6.059,149.140
C01049=1158.891,1.306,-47.145,179.828,6.060,149.140
C01050=1158.885,1.576,-47.159,179.830,6.060,149.139
C01051=1158.880,1.845,-47.174,179.833,6.061,149.138
C01052=1158.874,2.114,-47.188,179.836,6.063,149.138
C01053=1158.868,2.384,-47.203,179.839,6.063,149.137
C01054=1158.864,2.634,-47.216,179.841,6.063,149.136
C01055=1158.858,2.883,-47.230,179.843,6.064,149.136
C01056=1158.853,3.133,-47.244,179.846,6.065,149.135
C01057=1158.848,3.382,-47.256,179.848,6.066,149.135
C01058=1158.843,3.632,-47.271,179.851,6.066,149.134
C01059=1158.837,3.882,-47.284,179.854,6.068,149.134
C01060=1158.833,4.131,-47.298,179.856,6.068,149.133
C01061=1158.827,4.381,-47.311,179.858,6.069,149.132
C01062=1158.823,4.630,-47.325,179.861,6.069,149.132
C01063=1158.817,4.880,-47.338,179.863,6.070,149.131
C01064=1158.812,5.129,-47.352,179.866,6.071,149.131
C01065=1158.808,5.379,-47.365,179.868,6.071,149.130
C01066=1158.802,5.628,-47.379,179.871,6.072,149.129
C01067=1158.797,5.878,-47.393,179.874,6.074,149.129
C01068=1158.792,6.127,-47.406,179.876,6.074,149.128
C01069=1158.787,6.377,-47.420,179.878,6.075,149.128
C01070=1158.781,6.627,-47.433,179.881,6.075,149.127
C01071=1158.776,6.876,-47.447,179.884,6.076,149.126
C01072=1158.772,7.127,-47.460,179.886,6.077,149.126
C01073=1158.766,7.376,-47.474,179.888,6.077,149.125
C01074=1158.761,7.625,-47.489,179.891,6.079,149.125
C01075=1158.756,7.875,-47.501,179.894,6.079,149.124
C01076=1158.751,8.124,-47.516,179.896,6.080,149.124
C01077=1158.746,8.374,-47.530,179.899,6.080,149.123
C01078=1158.740,8.624,-47.543,179.901,6.081,149.123
C01079=1158.736,8.873,-47.557,179.904,6.082,149.122
C01080=1158.731,9.122,-47.571,179.906,6.082,149.121
C01081=1158.725,9.372,-47.584,179.909,6.084,149.121
C01082=1158.720,9.622,-47.598,179.911,6.085,149.120
C01083=1158.716,9.871,-47.612,179.914,6.085,149.120
C01084=1158.710,10.121,-47.625,179.916,6.086,149.119
C01085=1158.705,10.371,-47.640,179.919,6.086,149.118
C01086=1158.700,10.620,-47.653,179.921,6.087,149.118
C01087=1158.695,10.870,-47.668,179.924,6.088,149.117
C01088=1158.690,11.119,-47.680,179.926,6.089,149.117
C01089=1158.685,11.369,-47.695,179.929,6.090,149.116
C01090=1158.680,11.618,-47.709,179.931,6.090,149.115
C01091=1158.674,11.867,-47.723,179.934,6.091,149.115
C01092=1158.669,12.118,-47.736,179.936,6.091,149.114
C01093=1158.664,12.367,-47.751,179.939,6.093,149.114
C01094=1158.659,12.616,-47.764,179.942,6.093,149.113
C01095=1158.654,12.866,-47.778,179.944,6.094,149.113
C01096=1158.649,13.115,-47.793,179.947,6.095,149.112
C01097=1158.644,13.366,-47.806,179.949,6.096,149.112
C01098=1158.639,13.615,-47.820,179.951,6.096,149.111
C01099=1158.634,13.864,-47.834,179.954,6.098,149.110
C01100=1158.629,14.114,-47.849,179.957,6.098,149.110
C01101=1158.624,14.363,-47.862,179.959,6.099,149.109
C01102=1158.619,14.613,-47.876,179.962,6.099,149.109
C01103=1158.614,14.862,-47.890,179.964,6.100,149.108
C01104=1158.608,15.112,-47.904,179.967,6.102,149.107
C01105=1158.603,15.362,-47.918,179.969,6.102,149.107
C01106=1158.598,15.611,-47.932,179.972,6.103,149.106
C01107=1158.593,15.861,-47.946,179.974,6.104,149.106
C01108=1158.588,16.110,-47.960,179.977,6.104,149.105
C01109=1158.583,16.360,-47.975,179.979,6.106,149.105
C01110=1158.578,16.609,-47.989,179.982,6.106,149.104
C01111=1158.573,16.859,-48.003,179.984,6.107,149.104
C01112=1158.567,17.108,-48.017,179.987,6.108,149.103
C01113=1158.562,17.358,-48.031,179.990,6.108,149.102
C01114=1158.558,17.607,-48.045,179.992,6.110,149.102
C01115=1158.553,17.857,-48.059,179.995,6.110,149.101
C01116=1158.548,18.106,-48.073,179.997,6.111,149.101
C01117=1158.543,18.356,-48.088,180.000,6.111,149.100
C01118=1158.538,18.605,-48.102,-179.998,6.112,149.100
C01119=1158.533,18.855,-48.116,-179.995,6.113,149.099
C01120=1158.528,19.105,-48.130,-179.993,6.114,149.098
C01121=1158.522,19.354,-48.144,-179.990,6.115,149.098
C01122=1158.517,19.604,-48.159,-179.988,6.116,149.097
C01123=1158.512,19.853,-48.173,-179.985,6.117,149.097
C01124=1158.507,20.103,-48.187,-179.982,6.118,149.096
C01125=1158.502,20.353,-48.201,-179.980,6.118,149.095
C01126=1158.496,20.602,-48.216,-179.978,6.119,149.095
C01127=1158.491,20.852,-48.230,-179.975,6.119,149.094
C01128=1158.486,21.101,-48.244,-179.972,6.121,149.094
C01129=1158.481,21.351,-48.259,-179.970,6.122,149.093
C01130=1158.477,21.600,-48.274,-179.967,6.122,149.093
C01131=1158.471,21.849,-48.288,-179.965,6.123,149.092
C01132=1158.466,22.099,-48.302,-179.962,6.124,149.092
C01133=1158.461,22.349,-48.316,-179.959,6.125,149.091
C01134=1158.456,22.598,-48.330,-179.957,6.126,149.090
C01135=1158.451,22.848,-48.345,-179.955,6.126,149.090
C01136=1158.446,23.098,-48.359,-179.952,6.128,149.089
C01137=1158.441,23.346,-48.374,-179.949,6.128,149.089
C01138=1158.436,23.596,-48.388,-179.947,6.129,149.088
C01139=1158.430,23.846,-48.403,-179.944,6.130,149.087
C01140=1158.425,24.096,-48.417,-179.942,6.131,149.087
C01141=1158.420,24.345,-48.431,-179.939,6.132,149.086
C01142=1158.416,24.594,-48.446,-179.937,6.133,149.086
C01143=1158.411,24.844,-48.461,-179.934,6.133,149.085
C01144=1158.406,25.094,-48.475,-179.932,6.134,149.085
C01145=1158.400,25.343,-48.489,-179.929,6.135,149.084
C01146=1158.395,25.592,-48.504,-179.927,6.136,149.084
C01147=1158.390,25.842,-48.519,-179.924,6.136,149.083
C01148=1158.385,26.092,-48.533,-179.921,6.138,149.082
C01149=1158.380,26.341,-48.547,-179.918,6.139,149.082
C01150=1158.375,26.591,-48.562,-179.916,6.139,149.081
C01151=1158.370,26.840,-48.577,-179.914,6.140,149.081
C01152=1158.365,27.090,-48.591,-179.911,6.142,149.080
C01153=1158.360,27.339,-48.606,-179.908,6.142,149.080
C01154=1158.355,27.609,-48.621,-179.906,6.142,149.079
C01155=1158.349,27.878,-48.638,-179.903,6.144,149.078
C01156=1158.343,28.146,-48.653,-179.900,6.145,149.078
C01157=1158.338,28.415,-48.669,-179.897,6.146,149.077
C01158=1158.333,28.664,-48.683,-179.895,6.147,149.077
C01159=1158.328,28.914,-48.699,-179.892,6.147,149.076
C01160=1158.323,29.164,-48.713,-179.890,6.148,149.075
C01161=1158.318,29.413,-48.728,-179.887,6.149,149.075
C01162=1158.313,29.662,-48.742,-179.885,6.150,149.074
C01163=1158.307,29.912,-48.757,-179.882,6.151,149.074
C01164=1158.303,30.161,-48.772,-179.879,6.152,149.073
C01165=1158.298,30.411,-48.786,-179.877,6.153,149.073
C01166=1158.292,30.661,-48.802,-179.874,6.154,149.072
C01167=1158.287,30.910,-48.816,-179.872,6.154,149.071
C01168=1158.283,31.159,-48.831,-179.869,6.156,149.071
C01169=1158.278,31.409,-48.845,-179.866,6.156,149.070
C01170=1158.272,31.659,-48.860,-179.864,6.157,149.070
C01171=1158.267,31.908,-48.875,-179.861,6.158,149.069
C01172=1158.263,32.158,-48.890,-179.859,6.159,149.069
C01173=1158.257,32.407,-48.905,-179.856,6.160,149.068
C01174=1158.252,32.657,-48.919,-179.853,6.161,149.068
C01175=1158.248,32.906,-48.934,-179.851,6.162,149.067
C01176=1158.242,33.156,-48.950,-179.849,6.163,149.066
C01177=1158.237,33.405,-48.964,-179.846,6.163,149.066
C01178=1158.232,33.655,-48.980,-179.843,6.165,149.065
C01179=1158.227,33.904,-48.994,-179.841,6.165,149.065
C01180=1158.222,34.153,-49.009,-179.838,6.166,149.064
C01181=1158.217,34.403,-49.024,-179.835,6.167,149.064
C01182=1158.212,34.653,-49.039,-179.833,6.168,149.063
C01183=1158.207,34.902,-49.053,-179.830,6.169,149.062
C01184=1158.202,35.152,-49.069,-179.828,6.170,149.062
C01185=1158.197,35.401,-49.084,-179.825,6.171,149.061
C01186=1158.191,35.651,-49.099,-179.823,6.172,149.061
C01187=1158.187,35.900,-49.114,-179.820,6.173,149.060
C01188=1158.182,36.150,-49.130,-179.817,6.174,149.060
C01189=1158.177,36.400,-49.144,-179.815,6.175,149.059
C01190=1158.172,36.649,-49.159,-179.812,6.176,149.059
C01191=1158.167,36.898,-49.175,-179.810,6.177,149.058
C01192=1158.162,37.148,-49.189,-179.807,6.177,149.057
C01193=1158.156,37.397,-49.204,-179.804,6.179,149.057
C01194=1158.152,37.646,-49.219,-179.802,6.179,149.056
C01195=1158.146,37.896,-49.234,-179.800,6.180,149.056
C01196=1158.141,38.146,-49.249,-179.796,6.181,149.055
C01197=1158.136,38.395,-49.265,-179.794,6.182,149.055
C01198=1158.131,38.645,-49.279,-179.792,6.183,149.054
C01199=1158.126,38.894,-49.295,-179.789,6.184,149.054
C01200=1158.122,39.144,-49.310,-179.786,6.185,149.053
C01201=1158.116,39.393,-49.326,-179.784,6.186,149.053
C01202=1158.111,39.643,-49.340,-179.781,6.187,149.052
C01203=1158.106,39.892,-49.356,-179.779,6.188,149.051
C01204=1158.101,40.141,-49.370,-179.776,6.188,149.051
C01205=1158.096,40.391,-49.386,-179.773,6.190,149.050
C01206=1158.090,40.640,-49.402,-179.771,6.190,149.050
C01207=1158.086,40.891,-49.416,-179.768,6.191,149.049
C01208=1158.081,41.140,-49.432,-179.765,6.193,149.048
C01209=1158.076,41.389,-49.447,-179.763,6.193,149.048
C01210=1158.071,41.639,-49.462,-179.760,6.194,149.047
C01211=1158.066,41.888,-49.477,-179.758,6.196,149.047
C01212=1158.061,42.137,-49.493,-179.755,6.196,149.046
C01213=1158.056,42.388,-49.508,-179.753,6.197,149.046
C01214=1158.051,42.637,-49.523,-179.750,6.199,149.045
C01215=1158.046,42.886,-49.539,-179.747,6.199,149.045
C01216=1158.041,43.135,-49.554,-179.745,6.201,149.044
C01217=1158.036,43.385,-49.569,-179.742,6.201,149.044
C01218=1158.030,43.634,-49.585,-179.740,6.202,149.043
C01219=1158.026,43.884,-49.600,-179.737,6.203,149.042
C01220=1158.021,44.133,-49.616,-179.734,6.204,149.042
C01221=1158.016,44.382,-49.631,-179.732,6.205,149.041
C01222=1158.011,44.632,-49.647,-179.729,6.206,149.041
C01223=1158.005,44.881,-49.662,-179.726,6.207,149.040
C01224=1158.001,45.131,-49.678,-179.724,6.208,149.040
C01225=1157.996,45.380,-49.693,-179.721,6.209,149.039
C01226=1157.990,45.630,-49.709,-179.719,6.210,149.039
C01227=1157.986,45.879,-49.724,-179.716,6.211,149.038
C01228=1157.981,46.129,-49.740,-179.714,6.212,149.038
C01229=1157.976,46.378,-49.755,-179.711,6.213,149.037
C01230=1157.970,46.628,-49.771,-179.708,6.214,149.036
C01231=1157.966,46.877,-49.786,-179.706,6.215,149.036
C01232=1157.961,47.127,-49.802,-179.703,6.216,149.035
C01233=1157.955,47.376,-49.817,-179.701,6.217,149.035
C01234=1157.951,47.626,-49.832,-179.698,6.217,149.034
C01235=1157.945,47.875,-49.848,-179.695,6.219,149.034
C01236=1157.941,48.125,-49.864,-179.693,6.220,149.033
C01237=1157.935,48.374,-49.879,-179.690,6.221,149.033
C01238=1157.931,48.624,-49.894,-179.688,6.222,149.032
C01239=1157.926,48.874,-49.910,-179.685,6.223,149.032
C01240=1157.920,49.123,-49.926,-179.682,6.224,149.031
C01241=1157.915,49.372,-49.942,-179.680,6.225,149.030
C01242=1157.911,49.621,-49.957,-179.677,6.226,149.030
C01243=1157.906,49.871,-49.973,-179.674,6.227,149.029
C01244=1157.900,50.120,-49.989,-179.671,6.229,149.029
C01245=1157.895,50.370,-50.004,-179.669,6.229,149.028
C01246=1157.890,50.620,-50.020,-179.667,6.230,149.028
C01247=1157.886,50.869,-50.035,-179.663,6.231,149.027
C01248=1157.881,51.118,-50.052,-179.661,6.232,149.027
C01249=1157.876,51.368,-50.068,-179.659,6.234,149.026
C01250=1157.870,51.617,-50.083,-179.656,6.234,149.026
C01251=1157.865,51.867,-50.099,-179.654,6.235,149.025
C01252=1157.861,52.116,-50.115,-179.651,6.236,149.024
C01253=1157.856,52.365,-50.130,-179.648,6.237,149.024
C01254=1157.851,52.615,-50.146,-179.645,6.238,149.023
C01255=1157.846,52.865,-50.162,-179.643,6.239,149.023
C01256=1157.841,53.114,-50.178,-179.640,6.241,149.022
C01257=1157.836,53.364,-50.194,-179.638,6.242,149.022
C01258=1157.830,53.632,-50.211,-179.634,6.243,149.021
C01259=1157.825,53.901,-50.228,-179.632,6.244,149.021
C01260=1157.819,54.169,-50.245,-179.629,6.245,149.020
C01261=1157.814,54.438,-50.262,-179.626,6.247,149.020
C01262=1157.809,54.688,-50.278,-179.624,6.247,149.019
C01263=1157.804,54.936,-50.295,-179.621,6.248,149.018
C01264=1157.800,55.186,-50.310,-179.618,6.249,149.018
C01265=1157.794,55.436,-50.326,-179.616,6.250,149.017
C01266=1157.789,55.684,-50.342,-179.613,6.251,149.017
C01267=1157.784,55.935,-50.358,-179.611,6.252,149.016
C01268=1157.779,56.183,-50.374,-179.608,6.254,149.016
C01269=1157.775,56.433,-50.390,-179.605,6.254,149.015
C01270=1157.769,56.683,-50.406,-179.603,6.256,149.015
C01271=1157.764,56.932,-50.422,-179.600,6.257,149.014
C01272=1157.759,57.182,-50.438,-179.597,6.258,149.014
C01273=1157.754,57.430,-50.454,-179.595,6.259,149.013
C01274=1157.749,57.681,-50.470,-179.592,6.260,149.012
C01275=1157.744,57.929,-50.486,-179.590,6.261,149.012
C01276=1157.740,58.179,-50.502,-179.587,6.262,149.011
C01277=1157.734,58.429,-50.518,-179.584,6.263,149.011
C01278=1157.730,58.678,-50.535,-179.582,6.264,149.010
C01279=1157.724,58.928,-50.550,-179.579,6.266,149.010
C01280=1157.719,59.177,-50.567,-179.576,6.266,149.009
C01281=1157.714,59.427,-50.583,-179.574,6.268,149.009
C01282=1157.709,59.675,-50.599,-179.571,6.269,149.008
C01283=1157.705,59.926,-50.615,-179.568,6.270,149.008
C01284=1157.700,60.174,-50.631,-179.566,6.271,149.007
C01285=1157.694,60.424,-50.648,-179.563,6.272,149.007
C01286=1157.689,60.674,-50.664,-179.561,6.273,149.006
C01287=1157.684,60.923,-50.681,-179.557,6.274,149.005
C01288=1157.679,61.172,-50.696,-179.555,6.275,149.005
C01289=1157.675,61.422,-50.713,-179.552,6.277,149.005
C01290=1157.669,61.671,-50.728,-179.550,6.277,149.004
C01291=1157.665,61.921,-50.745,-179.547,6.279,149.003
C01292=1157.660,62.170,-50.761,-179.544,6.279,149.003
C01293=1157.655,62.420,-50.777,-179.542,6.281,149.002
C01294=1157.650,62.668,-50.794,-179.540,6.282,149.002
C01295=1157.645,62.918,-50.811,-179.536,6.283,149.001
C01296=1157.640,63.168,-50.827,-179.534,6.284,149.001
C01297=1157.635,63.417,-50.843,-179.531,6.285,149.000
C01298=1157.630,63.667,-50.860,-179.529,6.286,149.000
C01299=1157.625,63.916,-50.875,-179.526,6.288,148.999
C01300=1157.620,64.166,-50.892,-179.523,6.288,148.999
C01301=1157.615,64.414,-50.908,-179.521,6.290,148.998
C01302=1157.610,64.665,-50.925,-179.518,6.291,148.998
C01303=1157.605,64.913,-50.941,-179.515,6.292,148.997
C01304=1157.600,65.163,-50.958,-179.513,6.293,148.997
C01305=1157.596,65.412,-50.975,-179.510,6.294,148.996
C01306=1157.590,65.662,-50.990,-179.508,6.295,148.996
C01307=1157.585,65.912,-51.007,-179.505,6.297,148.995
C01308=1157.580,66.160,-51.024,-179.502,6.297,148.994
C01309=1157.576,66.410,-51.040,-179.500,6.299,148.994
C01310=1157.571,66.660,-51.056,-179.497,6.300,148.993
C01311=1157.565,66.909,-51.073,-179.494,6.301,148.993
C01312=1157.560,67.159,-51.090,-179.492,6.302,148.992
C01313=1157.555,67.407,-51.106,-179.489,6.303,148.992
C01314=1157.551,67.657,-51.123,-179.487,6.304,148.991
C01315=1157.546,67.907,-51.140,-179.484,6.306,148.991
C01316=1157.540,68.156,-51.156,-179.481,6.307,148.990
C01317=1157.536,68.406,-51.172,-179.478,6.308,148.990
C01318=1157.531,68.655,-51.189,-179.475,6.310,148.989
C01319=1157.526,68.904,-51.206,-179.473,6.310,148.989
C01320=1157.521,69.154,-51.223,-179.470,6.312,148.988
C01321=1157.516,69.402,-51.239,-179.468,6.313,148.988
C01322=1157.511,69.652,-51.256,-179.465,6.314,148.987
C01323=1157.506,69.902,-51.273,-179.463,6.315,148.987
C01324=1157.501,70.150,-51.289,-179.460,6.316,148.986
C01325=1157.496,70.400,-51.307,-179.457,6.317,148.986
C01326=1157.491,70.650,-51.322,-179.454,6.319,148.985
C01327=1157.486,70.899,-51.339,-179.452,6.319,148.985
C01328=1157.481,71.149,-51.356,-179.449,6.321,148.984
C01329=1157.476,71.398,-51.373,-179.446,6.322,148.984
C01330=1157.471,71.647,-51.389,-179.444,6.323,148.983
C01331=1157.466,71.897,-51.406,-179.441,6.325,148.983
C01332=1157.462,72.146,-51.423,-179.439,6.325,148.982
C01333=1157.457,72.396,-51.440,-179.436,6.327,148.981
C01334=1157.451,72.645,-51.456,-179.433,6.328,148.981
C01335=1157.447,72.895,-51.473,-179.431,6.329,148.981
C01336=1157.442,73.144,-51.490,-179.427,6.331,148.980
C01337=1157.437,73.392,-51.507,-179.425,6.332,148.979
C01338=1157.432,73.642,-51.525,-179.422,6.333,148.979
C01339=1157.427,73.892,-51.541,-179.420,6.334,148.978
C01340=1157.423,74.141,-51.558,-179.417,6.335,148.978
C01341=1157.417,74.390,-51.575,-179.415,6.336,148.977
C01342=1157.412,74.640,-51.592,-179.412,6.338,148.977
C01343=1157.407,74.890,-51.609,-179.409,6.339,148.976
C01344=1157.403,75.139,-51.626,-179.407,6.340,148.976
C01345=1157.397,75.388,-51.642,-179.404,6.341,148.975
C01346=1157.392,75.638,-51.659,-179.401,6.342,148.975
C01347=1157.387,75.887,-51.677,-179.398,6.344,148.974
C01348=1157.383,76.136,-51.694,-179.396,6.344,148.974
C01349=1157.377,76.385,-51.711,-179.393,6.346,148.973
C01350=1157.373,76.635,-51.727,-179.390,6.347,148.973
C01351=1157.367,76.885,-51.745,-179.388,6.348,148.972
C01352=1157.363,77.134,-51.762,-179.385,6.350,148.972
C01353=1157.358,77.383,-51.779,-179.383,6.351,148.971
C01354=1157.353,77.632,-51.796,-179.380,6.352,148.971
C01355=1157.348,77.882,-51.813,-179.377,6.354,148.970
C01356=1157.343,78.131,-51.829,-179.375,6.354,148.970
C01357=1157.338,78.381,-51.847,-179.372,6.356,148.969
C01358=1157.334,78.630,-51.864,-179.369,6.357,148.969
C01359=1157.328,78.879,-51.881,-179.367,6.358,148.968
C01360=1157.323,79.128,-51.899,-179.364,6.360,148.968
C01361=1157.319,79.378,-51.916,-179.361,6.360,148.967
C01362=1157.313,79.647,-51.934,-179.358,6.362,148.967
C01363=1157.307,79.915,-51.953,-179.355,6.363,148.966
C01364=1157.303,80.183,-51.971,-179.353,6.365,148.966
C01365=1157.298,80.452,-51.990,-179.349,6.366,148.965
C01366=1157.292,80.701,-52.007,-179.347,6.367,148.965
C01367=1157.287,80.950,-52.024,-179.344,6.369,148.964
C01368=1157.282,81.199,-52.042,-179.342,6.370,148.963
C01369=1157.278,81.449,-52.058,-179.339,6.371,148.963
C01370=1157.273,81.699,-52.076,-179.336,6.373,148.962
C01371=1157.268,81.948,-52.094,-179.334,6.373,148.962
C01372=1157.263,82.197,-52.110,-179.331,6.375,148.962
C01373=1157.258,82.447,-52.128,-179.328,6.376,148.961
C01374=1157.253,82.696,-52.145,-179.326,6.377,148.960
C01375=1157.248,82.945,-52.163,-179.323,6.379,148.960
C01376=1157.243,83.194,-52.180,-179.320,6.379,148.959
C01377=1157.238,83.444,-52.197,-179.318,6.381,148.959
C01378=1157.234,83.693,-52.215,-179.315,6.383,148.959
C01379=1157.229,83.943,-52.232,-179.312,6.383,148.958
C01380=1157.224,84.192,-52.250,-179.309,6.385,148.957
C01381=1157.218,84.442,-52.267,-179.307,6.387,148.957
C01382=1157.214,84.691,-52.284,-179.304,6.387,148.956
C01383=1157.209,84.940,-52.302,-179.301,6.389,148.956
C01384=1157.204,85.190,-52.320,-179.299,6.391,148.956
C01385=1157.199,85.439,-52.337,-179.296,6.391,148.955
C01386=1157.194,85.688,-52.354,-179.293,6.393,148.954
C01387=1157.189,85.937,-52.372,-179.291,6.394,148.954
C01388=1157.184,86.187,-52.389,-179.288,6.395,148.954
C01389=1157.179,86.436,-52.407,-179.285,6.397,148.953
C01390=1157.175,86.685,-52.424,-179.282,6.398,148.953
C01391=1157.170,86.934,-52.442,-179.280,6.399,148.952
C01392=1157.165,87.184,-52.460,-179.277,6.401,148.952
C01393=1157.160,87.433,-52.477,-179.274,6.402,148.951
C01394=1157.155,87.683,-52.495,-179.272,6.403,148.951
C01395=1157.150,87.932,-52.512,-179.269,6.404,148.950
C01396=1157.145,88.181,-52.530,-179.266,6.406,148.950
C01397=1157.140,88.430,-52.548,-179.264,6.407,148.949
C01398=1157.135,88.680,-52.565,-179.261,6.408,148.949
C01399=1157.130,88.929,-52.583,-179.258,6.410,148.948
C01400=1157.125,89.179,-52.601,-179.256,6.411,148.948
C01401=1157.120,89.428,-52.618,-179.253,6.413,148.947
C01402=1157.116,89.677,-52.636,-179.250,6.414,148.947
C01403=1157.111,89.926,-52.654,-179.248,6.415,148.946
C01404=1157.106,90.176,-52.672,-179.245,6.417,148.946
C01405=1157.101,90.425,-52.689,-179.242,6.418,148.945
C01406=1157.096,90.674,-52.707,-179.240,6.419,148.945
C01407=1157.091,90.924,-52.725,-179.237,6.420,148.944
C01408=1157.086,91.173,-52.743,-179.234,6.422,148.944
C01409=1157.081,91.423,-52.760,-179.231,6.423,148.943
C01410=1157.076,91.672,-52.778,-179.229,6.424,148.943
C01411=1157.072,91.922,-52.796,-179.226,6.426,148.942
C01412=1157.067,92.171,-52.814,-179.223,6.427,148.942
C01413=1157.063,92.420,-52.832,-179.221,6.428,148.941
C01414=1157.058,92.669,-52.850,-179.218,6.430,148.941
C01415=1157.052,92.919,-52.867,-179.215,6.431,148.940
C01416=1157.048,93.168,-52.885,-179.213,6.432,148.940
C01417=1157.043,93.417,-52.903,-179.210,6.434,148.939
C01418=1157.038,93.666,-52.921,-179.207,6.435,148.939
C01419=1157.033,93.915,-52.939,-179.204,6.437,148.938
C01420=1157.028,94.165,-52.957,-179.202,6.438,148.938
C01421=1157.023,94.414,-52.975,-179.199,6.439,148.938
C01422=1157.018,94.663,-52.993,-179.196,6.441,148.937
C01423=1157.014,94.913,-53.011,-179.194,6.442,148.936
C01424=1157.009,95.163,-53.028,-179.191,6.443,148.936
C01425=1157.004,95.412,-53.046,-179.189,6.445,148.936
C01426=1156.999,95.661,-53.064,-179.185,6.446,148.935
C01427=1156.994,95.910,-53.082,-179.183,6.447,148.935
C01428=1156.989,96.159,-53.100,-179.180,6.449,148.934
C01429=1156.983,96.409,-53.119,-179.178,6.451,148.934
C01430=1156.978,96.658,-53.137,-179.175,6.452,148.933
C01431=1156.974,96.908,-53.155,-179.172,6.453,148.933
C01432=1156.969,97.157,-53.173,-179.170,6.455,148.932
C01433=1156.964,97.406,-53.191,-179.166,6.456,148.932
C01434=1156.959,97.655,-53.209,-179.164,6.458,148.931
C01435=1156.954,97.905,-53.227,-179.162,6.458,148.931
C01436=1156.949,98.154,-53.245,-179.159,6.460,148.930
C01437=1156.945,98.403,-53.264,-179.156,6.461,148.930
C01438=1156.941,98.652,-53.282,-179.154,6.462,148.929
C01439=1156.935,98.902,-53.301,-179.151,6.464,148.929
C01440=1156.930,99.151,-53.319,-179.148,6.466,148.928
C01441=1156.925,99.400,-53.337,-179.145,6.467,148.928
C01442=1156.921,99.650,-53.355,-179.142,6.469,148.927
C01443=1156.916,99.899,-53.373,-179.140,6.470,148.927
C01444=1156.911,100.148,-53.391,-179.137,6.471,148.927
C01445=1156.906,100.397,-53.409,-179.134,6.473,148.926
C01446=1156.901,100.646,-53.428,-179.131,6.474,148.926
C01447=1156.896,100.896,-53.447,-179.129,6.475,148.925
C01448=1156.891,101.145,-53.465,-179.126,6.477,148.925
C01449=1156.887,101.394,-53.483,-179.123,6.478,148.924
C01450=1156.882,101.644,-53.501,-179.121,6.480,148.924
C01451=1156.877,101.893,-53.520,-179.118,6.481,148.923
C01452=1156.872,102.142,-53.538,-179.116,6.483,148.923
C01453=1156.867,102.392,-53.556,-179.112,6.484,148.922
C01454=1156.862,102.641,-53.574,-179.110,6.486,148.922
C01455=1156.857,102.890,-53.594,-179.108,6.486,148.921
C01456=1156.852,103.140,-53.612,-179.105,6.488,148.921
C01457=1156.848,103.389,-53.630,-179.102,6.490,148.920
C01458=1156.843,103.638,-53.648,-179.099,6.491,148.920
C01459=1156.838,103.887,-53.667,-179.096,6.493,148.919
C01460=1156.833,104.137,-53.685,-179.094,6.494,148.919
C01461=1156.828,104.386,-53.703,-179.091,6.496,148.919
C01462=1156.823,104.635,-53.723,-179.088,6.497,148.918
C01463=1156.818,104.885,-53.741,-179.085,6.499,148.918
C01464=1156.814,105.134,-53.759,-179.083,6.500,148.917
C01465=1156.809,105.382,-53.778,-179.081,6.501,148.917
C01466=1156.804,105.652,-53.798,-179.077,6.502,148.916
C01467=1156.799,105.920,-53.817,-179.075,6.504,148.916
C01468=1156.793,106.188,-53.838,-179.072,6.506,148.915
C01469=1156.788,106.456,-53.858,-179.069,6.507,148.915
C01470=1156.783,106.706,-53.876,-179.066,6.509,148.914
C01471=1156.778,106.955,-53.895,-179.063,6.511,148.914
C01472=1156.773,107.204,-53.914,-179.060,6.512,148.913
C01473=1156.769,107.453,-53.933,-179.057,6.514,148.913
C01474=1156.764,107.703,-53.951,-179.055,6.515,148.912
C01475=1156.758,107.951,-53.970,-179.052,6.516,148.912
C01476=1156.754,108.201,-53.988,-179.050,6.518,148.912
C01477=1156.749,108.450,-54.008,-179.047,6.519,148.911
C01478=1156.744,108.699,-54.026,-179.044,6.521,148.911
C01479=1156.740,108.949,-54.045,-179.041,6.523,148.910
C01480=1156.734,109.198,-54.063,-179.039,6.524,148.910
C01481=1156.730,109.447,-54.082,-179.036,6.525,148.909
C01482=1156.725,109.697,-54.101,-179.033,6.527,148.909
C01483=1156.720,109.945,-54.120,-179.030,6.528,148.908
C01484=1156.715,110.196,-54.139,-179.028,6.530,148.908
C01485=1156.710,110.444,-54.157,-179.025,6.532,148.907
C01486=1156.706,110.693,-54.176,-179.023,6.533,148.907
C01487=1156.701,110.943,-54.195,-179.020,6.534,148.906
C01488=1156.696,111.192,-54.214,-179.017,6.536,148.906
C01489=1156.691,111.442,-54.233,-179.014,6.537,148.906
C01490=1156.686,111.690,-54.251,-179.011,6.539,148.905
C01491=1156.682,111.940,-54.271,-179.009,6.541,148.905
C01492=1156.676,112.189,-54.290,-179.006,6.541,148.904
C01493=1156.672,112.439,-54.309,-179.003,6.543,148.904
C01494=1156.667,112.687,-54.328,-179.001,6.545,148.903
C01495=1156.662,112.937,-54.346,-178.998,6.546,148.903
C01496=1156.657,113.186,-54.366,-178.995,6.548,148.903
C01497=1156.652,113.435,-54.384,-178.992,6.550,148.902
C01498=1156.647,113.685,-54.403,-178.989,6.551,148.902
C01499=1156.643,113.933,-54.422,-178.987,6.552,148.901
C01500=1156.638,114.183,-54.441,-178.984,6.554,148.901
C01501=1156.633,114.432,-54.461,-178.982,6.556,148.900
C01502=1156.628,114.682,-54.479,-178.979,6.557,148.900
C01503=1156.623,114.931,-54.498,-178.976,6.559,148.899
C01504=1156.619,115.180,-54.517,-178.973,6.560,148.899
C01505=1156.614,115.429,-54.537,-178.970,6.562,148.898
C01506=1156.609,115.679,-54.556,-178.968,6.563,148.898
C01507=1156.604,115.928,-54.574,-178.965,6.565,148.898
C01508=1156.599,116.177,-54.594,-178.963,6.566,148.897
C01509=1156.595,116.426,-54.613,-178.960,6.568,148.897
C01510=1156.590,116.675,-54.632,-178.957,6.569,148.896
C01511=1156.585,116.924,-54.652,-178.954,6.571,148.896
C01512=1156.581,117.173,-54.671,-178.951,6.573,148.895
C01513=1156.575,117.423,-54.689,-178.949,6.574,148.895
C01514=1156.570,117.672,-54.709,-178.947,6.575,148.895
C01515=1156.565,117.921,-54.728,-178.944,6.577,148.894
C01516=1156.561,118.171,-54.747,-178.941,6.578,148.894
C01517=1156.555,118.419,-54.767,-178.938,6.580,148.893
C01518=1156.551,118.669,-54.786,-178.935,6.582,148.893
C01519=1156.547,118.918,-54.805,-178.932,6.584,148.892
C01520=1156.541,119.167,-54.825,-178.930,6.585,148.892
C01521=1156.537,119.417,-54.844,-178.927,6.587,148.892
C01522=1156.531,119.666,-54.864,-178.924,6.589,148.891
C01523=1156.527,119.915,-54.883,-178.922,6.589,148.890
C01524=1156.522,120.164,-54.902,-178.919,6.591,148.890
C01525=1156.517,120.413,-54.922,-178.916,6.593,148.890
C01526=1156.512,120.663,-54.941,-178.914,6.594,148.889
C01527=1156.508,120.911,-54.960,-178.911,6.596,148.889
C01528=1156.503,121.161,-54.980,-178.908,6.598,148.888
C01529=1156.498,121.410,-54.999,-178.905,6.599,148.888
C01530=1156.493,121.659,-55.019,-178.903,6.601,148.888
C01531=1156.489,121.909,-55.038,-178.900,6.603,148.887
C01532=1156.484,122.157,-55.057,-178.897,6.604,148.887
C01533=1156.479,122.407,-55.077,-178.894,6.606,148.886
C01534=1156.474,122.657,-55.096,-178.891,6.608,148.886
C01535=1156.469,122.905,-55.116,-178.889,6.609,148.885
C01536=1156.464,123.154,-55.136,-178.887,6.610,148.885
C01537=1156.460,123.404,-55.155,-178.884,6.612,148.885
C01538=1156.455,123.653,-55.174,-178.881,6.614,148.884
C01539=1156.450,123.902,-55.194,-178.878,6.615,148.884
C01540=1156.446,124.152,-55.214,-178.875,6.617,148.883
C01541=1156.440,124.401,-55.233,-178.872,6.618,148.883
C01542=1156.436,124.649,-55.253,-178.870,6.620,148.882
C01543=1156.431,124.899,-55.273,-178.867,6.622,148.882
C01544=1156.426,125.148,-55.292,-178.864,6.624,148.882
C01545=1156.422,125.397,-55.311,-178.862,6.625,148.881
C01546=1156.417,125.647,-55.331,-178.859,6.627,148.881
C01547=1156.412,125.895,-55.351,-178.856,6.629,148.880
C01548=1156.407,126.145,-55.371,-178.853,6.630,148.880
C01549=1156.402,126.394,-55.390,-178.850,6.632,148.879
C01550=1156.397,126.643,-55.409,-178.848,6.633,148.879
C01551=1156.393,126.892,-55.430,-178.845,6.634,148.879
C01552=1156.388,127.142,-55.450,-178.843,6.636,148.878
C01553=1156.383,127.391,-55.469,-178.840,6.638,148.878
C01554=1156.378,127.639,-55.489,-178.837,6.640,148.877
C01555=1156.373,127.889,-55.509,-178.835,6.641,148.877
C01556=1156.369,128.138,-55.528,-178.832,6.643,148.877
C01557=1156.364,128.387,-55.549,-178.829,6.645,148.876
C01558=1156.359,128.636,-55.568,-178.826,6.646,148.876
C01559=1156.354,128.886,-55.588,-178.823,6.648,148.875
C01560=1156.350,129.135,-55.608,-178.821,6.650,148.875
C01561=1156.345,129.384,-55.628,-178.818,6.651,148.874
C01562=1156.340,129.633,-55.648,-178.815,6.653,148.874
C01563=1156.335,129.882,-55.667,-178.812,6.655,148.874
C01564=1156.330,130.132,-55.687,-178.810,6.656,148.873
C01565=1156.326,130.381,-55.708,-178.807,6.658,148.873
C01566=1156.321,130.630,-55.727,-178.804,6.660,148.872
C01567=1156.316,130.879,-55.747,-178.802,6.662,148.872
C01568=1156.311,131.128,-55.767,-178.799,6.663,148.872
C01569=1156.307,131.377,-55.787,-178.796,6.665,148.871
C01570=1156.301,131.646,-55.809,-178.793,6.666,148.871
C01571=1156.296,131.915,-55.830,-178.790,6.668,148.870
C01572=1156.291,132.183,-55.852,-178.787,6.671,148.870
C01573=1156.286,132.452,-55.873,-178.784,6.672,148.870
C01574=1156.282,132.701,-55.894,-178.781,6.674,148.869
C01575=1156.276,132.949,-55.913,-178.779,6.676,148.869
C01576=1156.271,133.199,-55.934,-178.776,6.677,148.868
C01577=1156.266,133.448,-55.954,-178.773,6.679,148.868
C01578=1156.262,133.697,-55.974,-178.770,6.681,148.867
C01579=1156.258,133.946,-55.994,-178.767,6.682,148.867
C01580=1156.253,134.196,-56.014,-178.765,6.684,148.867
C01581=1156.248,134.444,-56.034,-178.762,6.686,148.866
C01582=1156.242,134.694,-56.054,-178.759,6.687,148.866
C01583=1156.238,134.943,-56.075,-178.757,6.689,148.865
C01584=1156.233,135.192,-56.095,-178.754,6.691,148.865
C01585=1156.229,135.441,-56.115,-178.751,6.693,148.865
C01586=1156.224,135.690,-56.135,-178.748,6.694,148.864
C01587=1156.219,135.940,-56.156,-178.746,6.696,148.864
C01588=1156.214,136.189,-56.176,-178.743,6.698,148.863
C01589=1156.210,136.438,-56.196,-178.740,6.699,148.863
C01590=1156.205,136.686,-56.216,-178.738,6.701,148.863
C01591=1156.200,136.936,-56.237,-178.735,6.703,148.862
C01592=1156.195,137.185,-56.257,-178.732,6.705,148.862
C01593=1156.191,137.434,-56.277,-178.730,6.706,148.861
C01594=1156.186,137.683,-56.298,-178.727,6.708,148.861
C01595=1156.181,137.932,-56.319,-178.724,6.710,148.861
C01596=1156.176,138.182,-56.338,-178.721,6.712,148.860
C01597=1156.172,138.431,-56.359,-178.719,6.713,148.860
C01598=1156.167,138.680,-56.380,-178.716,6.715,148.860
C01599=1156.162,138.929,-56.400,-178.713,6.717,148.859
C01600=1156.158,139.178,-56.420,-178.711,6.718,148.859
C01601=1156.153,139.427,-56.441,-178.708,6.720,148.858
C01602=1156.148,139.677,-56.461,-178.705,6.722,148.858
C01603=1156.143,139.926,-56.481,-178.702,6.724,148.858
C01604=1156.138,140.175,-56.502,-178.700,6.725,148.857
C01605=1156.134,140.424,-56.523,-178.696,6.728,148.857
C01606=1156.129,140.673,-56.543,-178.694,6.730,148.856
C01607=1156.124,140.922,-56.564,-178.691,6.731,148.856
C01608=1156.120,141.171,-56.584,-178.688,6.733,148.856
C01609=1156.115,141.420,-56.605,-178.686,6.735,148.855
C01610=1156.110,141.669,-56.626,-178.683,6.736,148.855
C01611=1156.106,141.918,-56.646,-178.680,6.738,148.854
C01612=1156.100,142.168,-56.667,-178.677,6.740,148.854
C01613=1156.096,142.416,-56.687,-178.675,6.742,148.854
C01614=1156.092,142.665,-56.708,-178.672,6.743,148.853
C01615=1156.086,142.915,-56.729,-178.669,6.745,148.853
C01616=1156.082,143.164,-56.749,-178.667,6.747,148.853
C01617=1156.077,143.413,-56.770,-178.664,6.749,148.852
C01618=1156.072,143.662,-56.790,-178.661,6.750,148.852
C01619=1156.067,143.911,-56.811,-178.659,6.752,148.851
C01620=1156.063,144.160,-56.832,-178.655,6.755,148.851
C01621=1156.058,144.409,-56.853,-178.653,6.756,148.851
C01622=1156.053,144.658,-56.873,-178.650,6.758,148.850
C01623=1156.048,144.908,-56.894,-178.647,6.760,148.850
C01624=1156.044,145.156,-56.914,-178.644,6.761,148.849
C01625=1156.038,145.406,-56.935,-178.642,6.763,148.849
C01626=1156.034,145.655,-56.956,-178.639,6.765,148.849
C01627=1156.029,145.904,-56.977,-178.636,6.767,148.848
C01628=1156.025,146.153,-56.998,-178.634,6.768,148.848
C01629=1156.020,146.402,-57.019,-178.631,6.770,148.848
C01630=1156.016,146.651,-57.040,-178.628,6.772,148.847
C01631=1156.010,146.900,-57.060,-178.625,6.774,148.847
C01632=1156.006,147.149,-57.081,-178.622,6.776,148.846
C01633=1156.001,147.398,-57.103,-178.619,6.778,148.846
C01634=1155.996,147.647,-57.123,-178.617,6.779,148.846
C01635=1155.992,147.896,-57.144,-178.614,6.781,148.845
C01636=1155.986,148.146,-57.165,-178.611,6.783,148.845
C01637=1155.983,148.395,-57.186,-178.609,6.785,148.844
C01638=1155.978,148.644,-57.207,-178.606,6.786,148.844
C01639=1155.972,148.893,-57.228,-178.603,6.788,148.844
C01640=1155.968,149.142,-57.249,-178.600,6.791,148.843
C01641=1155.963,149.391,-57.270,-178.597,6.792,148.843
C01642=1155.959,149.640,-57.291,-178.595,6.794,148.843
C01643=1155.954,149.889,-57.312,-178.592,6.796,148.842
C01644=1155.949,150.138,-57.334,-178.590,6.798,148.842
C01645=1155.945,150.387,-57.354,-178.587,6.800,148.842
C01646=1155.940,150.636,-57.375,-178.584,6.801,148.841
C01647=1155.935,150.885,-57.397,-178.582,6.803,148.841
C01648=1155.930,151.134,-57.417,-178.578,6.806,148.841
C01649=1155.926,151.384,-57.438,-178.576,6.807,148.840
C01650=1155.921,151.633,-57.460,-178.573,6.809,148.840
C01651=1155.916,151.882,-57.481,-178.570,6.811,148.839
C01652=1155.912,152.130,-57.502,-178.567,6.813,148.839
C01653=1155.906,152.379,-57.523,-178.565,6.814,148.839
C01654=1155.902,152.629,-57.544,-178.562,6.816,148.838
C01655=1155.897,152.878,-57.566,-178.559,6.819,148.838
C01656=1155.893,153.127,-57.586,-178.556,6.820,148.838
C01657=1155.888,153.376,-57.608,-178.553,6.822,148.837
C01658=1155.883,153.625,-57.629,-178.551,6.824,148.837
C01659=1155.878,153.874,-57.651,-178.548,6.826,148.837
C01660=1155.874,154.123,-57.672,-178.546,6.828,148.836
C01661=1155.869,154.372,-57.693,-178.543,6.829,148.836
C01662=1155.864,154.621,-57.714,-178.540,6.832,148.835
C01663=1155.859,154.870,-57.736,-178.537,6.834,148.835
C01664=1155.854,155.120,-57.757,-178.534,6.835,148.835
C01665=1155.850,155.368,-57.778,-178.532,6.837,148.834
C01666=1155.846,155.617,-57.800,-178.529,6.839,148.834
C01667=1155.841,155.867,-57.821,-178.526,6.841,148.834
C01668=1155.836,156.115,-57.843,-178.523,6.843,148.833
C01669=1155.831,156.365,-57.864,-178.521,6.845,148.833
C01670=1155.826,156.614,-57.886,-178.518,6.847,148.833
C01671=1155.822,156.862,-57.908,-178.515,6.849,148.832
C01672=1155.817,157.111,-57.928,-178.513,6.850,148.832
C01673=1155.813,157.361,-57.950,-178.510,6.852,148.832
C01674=1155.807,157.630,-57.973,-178.507,6.855,148.831
C01675=1155.802,157.898,-57.997,-178.504,6.856,148.831
C01676=1155.797,158.167,-58.020,-178.501,6.859,148.830
C01677=1155.792,158.436,-58.043,-178.498,6.861,148.830
C01678=1155.788,158.686,-58.065,-178.495,6.862,148.830
C01679=1155.783,158.934,-58.086,-178.492,6.865,148.829
C01680=1155.778,159.184,-58.107,-178.489,6.867,148.829
C01681=1155.774,159.433,-58.129,-178.487,6.868,148.829
C01682=1155.769,159.682,-58.151,-178.484,6.871,148.828
C01683=1155.764,159.930,-58.173,-178.482,6.872,148.828
C01684=1155.760,160.179,-58.195,-178.478,6.875,148.828
C01685=1155.754,160.429,-58.216,-178.476,6.877,148.827
C01686=1155.750,160.678,-58.238,-178.473,6.878,148.827
C01687=1155.745,160.927,-58.260,-178.470,6.880,148.827
C01688=1155.740,161.175,-58.281,-178.468,6.882,148.826
C01689=1155.736,161.425,-58.303,-178.465,6.885,148.826
C01690=1155.731,161.673,-58.325,-178.462,6.886,148.826
C01691=1155.727,161.923,-58.346,-178.459,6.888,148.825
C01692=1155.722,162.172,-58.368,-178.457,6.890,148.825
C01693=1155.717,162.421,-58.390,-178.454,6.892,148.825
C01694=1155.713,162.670,-58.412,-178.451,6.894,148.824
C01695=1155.708,162.919,-58.433,-178.448,6.896,148.824
C01696=1155.703,163.168,-58.455,-178.446,6.898,148.824
C01697=1155.699,163.417,-58.477,-178.443,6.900,148.823
C01698=1155.694,163.666,-58.499,-178.440,6.902,148.823
C01699=1155.689,163.915,-58.521,-178.437,6.904,148.823
C01700=1155.685,164.163,-58.543,-178.434,6.906,148.822
C01701=1155.680,164.413,-58.565,-178.432,6.907,148.822
C01702=1155.675,164.661,-58.587,-178.429,6.910,148.822
C01703=1155.670,164.911,-58.609,-178.426,6.912,148.821
C01704=1155.666,165.159,-58.631,-178.423,6.914,148.821
C01705=1155.661,165.409,-58.653,-178.421,6.916,148.821
C01706=1155.656,165.657,-58.674,-178.418,6.917,148.820
C01707=1155.652,165.907,-58.696,-178.415,6.920,148.820
C01708=1155.647,166.155,-58.718,-178.413,6.922,148.820
C01709=1155.642,166.405,-58.741,-178.410,6.924,148.819
C01710=1155.637,166.654,-58.762,-178.407,6.925,148.819
C01711=1155.633,166.903,-58.784,-178.404,6.928,148.819
C01712=1155.628,167.152,-58.806,-178.401,6.930,148.818
C01713=1155.624,167.400,-58.829,-178.399,6.932,148.818
C01714=1155.619,167.649,-58.851,-178.396,6.934,148.818
C01715=1155.614,167.899,-58.873,-178.393,6.936,148.817
C01716=1155.610,168.147,-58.895,-178.390,6.938,148.817
C01717=1155.605,168.397,-58.917,-178.388,6.940,148.817
C01718=1155.600,168.645,-58.939,-178.385,6.941,148.816
C01719=1155.596,168.894,-58.962,-178.382,6.944,148.816
C01720=1155.591,169.143,-58.984,-178.379,6.946,148.816
C01721=1155.587,169.392,-59.006,-178.377,6.948,148.815
C01722=1155.582,169.642,-59.028,-178.373,6.950,148.815
C01723=1155.577,169.890,-59.051,-178.371,6.952,148.815
C01724=1155.573,170.139,-59.073,-178.369,6.954,148.815
C01725=1155.568,170.388,-59.094,-178.366,6.956,148.814
C01726=1155.563,170.638,-59.117,-178.363,6.958,148.814
C01727=1155.558,170.886,-59.140,-178.360,6.960,148.813
C01728=1155.554,171.135,-59.162,-178.358,6.962,148.813
C01729=1155.549,171.385,-59.184,-178.355,6.964,148.813
C01730=1155.545,171.633,-59.207,-178.352,6.967,148.813
C01731=1155.540,171.882,-59.229,-178.349,6.968,148.812
C01732=1155.535,172.131,-59.251,-178.346,6.970,148.812
C01733=1155.531,172.380,-59.274,-178.344,6.973,148.812
C01734=1155.526,172.629,-59.296,-178.341,6.975,148.811
C01735=1155.521,172.878,-59.318,-178.338,6.976,148.811
C01736=1155.517,173.127,-59.341,-178.335,6.979,148.811
C01737=1155.511,173.376,-59.363,-178.333,6.981,148.811
C01738=1155.507,173.624,-59.386,-178.330,6.983,148.810
C01739=1155.503,173.874,-59.408,-178.327,6.985,148.810
C01740=1155.498,174.122,-59.431,-178.324,6.987,148.809
C01741=1155.493,174.371,-59.453,-178.322,6.989,148.809
C01742=1155.488,174.621,-59.476,-178.319,6.991,148.809
C01743=1155.484,174.869,-59.498,-178.316,6.994,148.809
C01744=1155.480,175.118,-59.520,-178.313,6.995,148.808
C01745=1155.475,175.367,-59.543,-178.311,6.997,148.808
C01746=1155.470,175.616,-59.565,-178.308,7.000,148.808
C01747=1155.465,175.865,-59.588,-178.305,7.002,148.807
C01748=1155.461,176.114,-59.611,-178.302,7.003,148.807
C01749=1155.456,176.363,-59.633,-178.299,7.006,148.807
C01750=1155.452,176.611,-59.656,-178.297,7.008,148.806
C01751=1155.447,176.861,-59.679,-178.294,7.010,148.806
C01752=1155.443,177.110,-59.702,-178.291,7.012,148.806
C01753=1155.437,177.359,-59.724,-178.289,7.014,148.806
C01754=1155.433,177.608,-59.747,-178.286,7.016,148.805
C01755=1155.429,177.857,-59.770,-178.283,7.019,148.805
C01756=1155.424,178.105,-59.792,-178.280,7.021,148.805
C01757=1155.419,178.354,-59.815,-178.278,7.023,148.804
C01758=1155.415,178.603,-59.838,-178.274,7.025,148.804
C01759=1155.410,178.853,-59.860,-178.272,7.027,148.804
C01760=1155.405,179.101,-59.883,-178.269,7.029,148.804
C01761=1155.401,179.350,-59.906,-178.266,7.032,148.803
C01762=1155.396,179.599,-59.929,-178.264,7.033,148.803
C01763=1155.392,179.848,-59.952,-178.261,7.035,148.803
C01764=1155.387,180.097,-59.975,-178.258,7.038,148.802
C01765=1155.382,180.345,-59.998,-178.255,7.040,148.802
C01766=1155.378,180.595,-60.020,-178.253,7.042,148.802
C01767=1155.373,180.844,-60.043,-178.250,7.044,148.802
C01768=1155.369,181.093,-60.066,-178.247,7.046,148.801
C01769=1155.364,181.341,-60.089,-178.244,7.048,148.801
C01770=1155.359,181.590,-60.113,-178.242,7.051,148.801
C01771=1155.355,181.839,-60.135,-178.239,7.053,148.800
C01772=1155.350,182.088,-60.158,-178.236,7.054,148.800
C01773=1155.345,182.337,-60.181,-178.234,7.057,148.800
C01774=1155.341,182.586,-60.204,-178.231,7.059,148.799
C01775=1155.336,182.834,-60.227,-178.228,7.062,148.799
C01776=1155.331,183.083,-60.250,-178.225,7.063,148.799
C01777=1155.327,183.332,-60.273,-178.223,7.065,148.799
C01778=1155.322,183.602,-60.298,-178.219,7.068,148.798
C01779=1155.317,183.872,-60.323,-178.216,7.071,148.798
C01780=1155.312,184.141,-60.348,-178.213,7.072,148.798
C01781=1155.307,184.411,-60.373,-178.211,7.075,148.797
C01782=1155.302,184.660,-60.396,-178.208,7.077,148.797
C01783=1155.297,184.909,-60.419,-178.205,7.079,148.797
C01784=1155.293,185.158,-60.442,-178.202,7.082,148.797
C01785=1155.289,185.407,-60.466,-178.199,7.084,148.796
C01786=1155.284,185.656,-60.489,-178.196,7.086,148.796
C01787=1155.279,185.905,-60.512,-178.194,7.088,148.796
C01788=1155.275,186.154,-60.536,-178.191,7.091,148.795
C01789=1155.270,186.402,-60.558,-178.188,7.092,148.795
C01790=1155.265,186.651,-60.581,-178.186,7.095,148.795
C01791=1155.261,186.900,-60.605,-178.183,7.097,148.795
C01792=1155.256,187.149,-60.628,-178.180,7.099,148.794
C01793=1155.252,187.397,-60.652,-178.177,7.102,148.794
C01794=1155.247,187.646,-60.676,-178.175,7.103,148.794
C01795=1155.243,187.895,-60.698,-178.171,7.106,148.793
C01796=1155.238,188.144,-60.722,-178.169,7.108,148.793
C01797=1155.233,188.393,-60.745,-178.167,7.110,148.793
C01798=1155.229,188.642,-60.768,-178.163,7.112,148.793
C01799=1155.224,188.891,-60.792,-178.161,7.114,148.793
C01800=1155.219,189.140,-60.815,-178.158,7.117,148.792
C01801=1155.215,189.389,-60.839,-178.156,7.119,148.792
C01802=1155.210,189.638,-60.863,-178.153,7.121,148.792
C01803=1155.205,189.886,-60.886,-178.150,7.123,148.791
C01804=1155.200,190.135,-60.909,-178.147,7.126,148.791
C01805=1155.197,190.383,-60.932,-178.144,7.128,148.791
C01806=1155.192,190.632,-60.956,-178.141,7.130,148.791
C01807=1155.187,190.881,-60.979,-178.139,7.133,148.790
C01808=1155.183,191.130,-61.002,-178.136,7.135,148.790
C01809=1155.178,191.379,-61.027,-178.134,7.137,148.790
C01810=1155.173,191.628,-61.050,-178.130,7.139,148.790
C01811=1155.169,191.877,-61.073,-178.128,7.141,148.789
C01812=1155.164,192.126,-61.097,-178.125,7.144,148.789
C01813=1155.160,192.374,-61.121,-178.122,7.146,148.789
C01814=1155.155,192.623,-61.144,-178.119,7.149,148.789
C01815=1155.151,192.872,-61.168,-178.117,7.150,148.788
C01816=1155.146,193.121,-61.191,-178.114,7.153,148.788
C01817=1155.142,193.370,-61.215,-178.111,7.155,148.788
C01818=1155.137,193.619,-61.239,-178.109,7.157,148.787
C01819=1155.133,193.868,-61.263,-178.106,7.160,148.787
C01820=1155.127,194.117,-61.287,-178.103,7.161,148.787
C01821=1155.123,194.366,-61.311,-178.100,7.164,148.787
C01822=1155.118,194.615,-61.334,-178.098,7.166,148.787
C01823=1155.114,194.863,-61.358,-178.094,7.169,148.786
C01824=1155.109,195.112,-61.381,-178.092,7.171,148.786
C01825=1155.105,195.360,-61.406,-178.089,7.173,148.786
C01826=1155.100,195.609,-61.429,-178.087,7.175,148.786
C01827=1155.096,195.858,-61.453,-178.083,7.178,148.785
C01828=1155.091,196.107,-61.476,-178.081,7.180,148.785
C01829=1155.086,196.355,-61.500,-178.078,7.183,148.785
C01830=1155.082,196.605,-61.525,-178.075,7.184,148.784
C01831=1155.077,196.854,-61.549,-178.073,7.187,148.784
C01832=1155.072,197.103,-61.572,-178.070,7.189,148.784
C01833=1155.068,197.351,-61.596,-178.068,7.191,148.784
C01834=1155.064,197.600,-61.620,-178.064,7.194,148.784
C01835=1155.059,197.849,-61.644,-178.062,7.196,148.783
